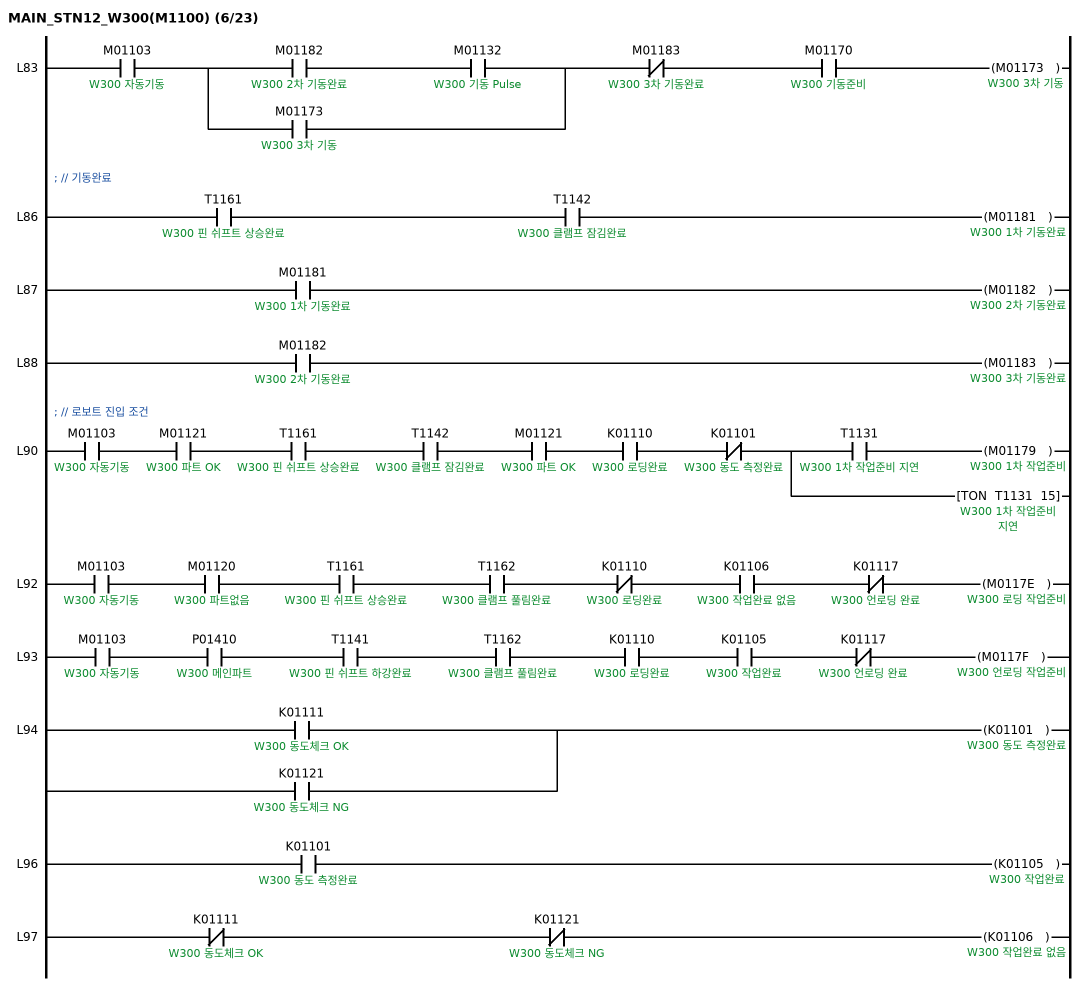
[picture p192: MAIN_STN12_W300(M1100) rungs L83-L97]
; L83
LOAD      M01103	// W300 자동기동
LOAD      M01182	// W300 2차 기동완료
AND       M01132	// W300 기동 Pulse
OR        M01173	// W300 3차 기동
AND LOAD
AND NOT   M01183	// W300 3차 기동완료
AND       M01170	// W300 기동준비
OUT       M01173	// W300 3차 기동
//   // 기동완료
; L86
LOAD      T1161	// W300 핀 쉬프트 상승완료
AND       T1142	// W300 클램프 잠김완료
OUT       M01181	// W300 1차 기동완료
; L87
LOAD      M01181	// W300 1차 기동완료
OUT       M01182	// W300 2차 기동완료
; L88
LOAD      M01182	// W300 2차 기동완료
OUT       M01183	// W300 3차 기동완료
//   // 로보트 진입 조건
; L90
LOAD      M01103	// W300 자동기동
AND       M01121	// W300 파트 OK
AND       T1161	// W300 핀 쉬프트 상승완료
AND       T1142	// W300 클램프 잠김완료
AND       M01121	// W300 파트 OK
AND       K01110	// W300 로딩완료
AND NOT   K01101	// W300 동도 측정완료
MPUSH
AND       T1131	// W300 1차 작업준비 지연
OUT       M01179	// W300 1차 작업준비
MPOP
TON       T1131 15	// W300 1차 작업준비 지연
; L92
LOAD      M01103	// W300 자동기동
AND       M01120	// W300 파트없음
AND       T1161	// W300 핀 쉬프트 상승완료
AND       T1162	// W300 클램프 풀림완료
AND NOT   K01110	// W300 로딩완료
AND       K01106	// W300 작업완료 없음
AND NOT   K01117	// W300 언로딩 완료
OUT       M0117E	// W300 로딩 작업준비
; L93
LOAD      M01103	// W300 자동기동
AND       P01410	// W300 메인파트
AND       T1141	// W300 핀 쉬프트 하강완료
AND       T1162	// W300 클램프 풀림완료
AND       K01110	// W300 로딩완료
AND       K01105	// W300 작업완료
AND NOT   K01117	// W300 언로딩 완료
OUT       M0117F	// W300 언로딩 작업준비
; L94
LOAD      K01111	// W300 동도체크 OK
OR        K01121	// W300 동도체크 NG
OUT       K01101	// W300 동도 측정완료
; L96
LOAD      K01101	// W300 동도 측정완료
OUT       K01105	// W300 작업완료
; L97
LOAD NOT  K01111	// W300 동도체크 OK
AND NOT   K01121	// W300 동도체크 NG
OUT       K01106	// W300 작업완료 없음

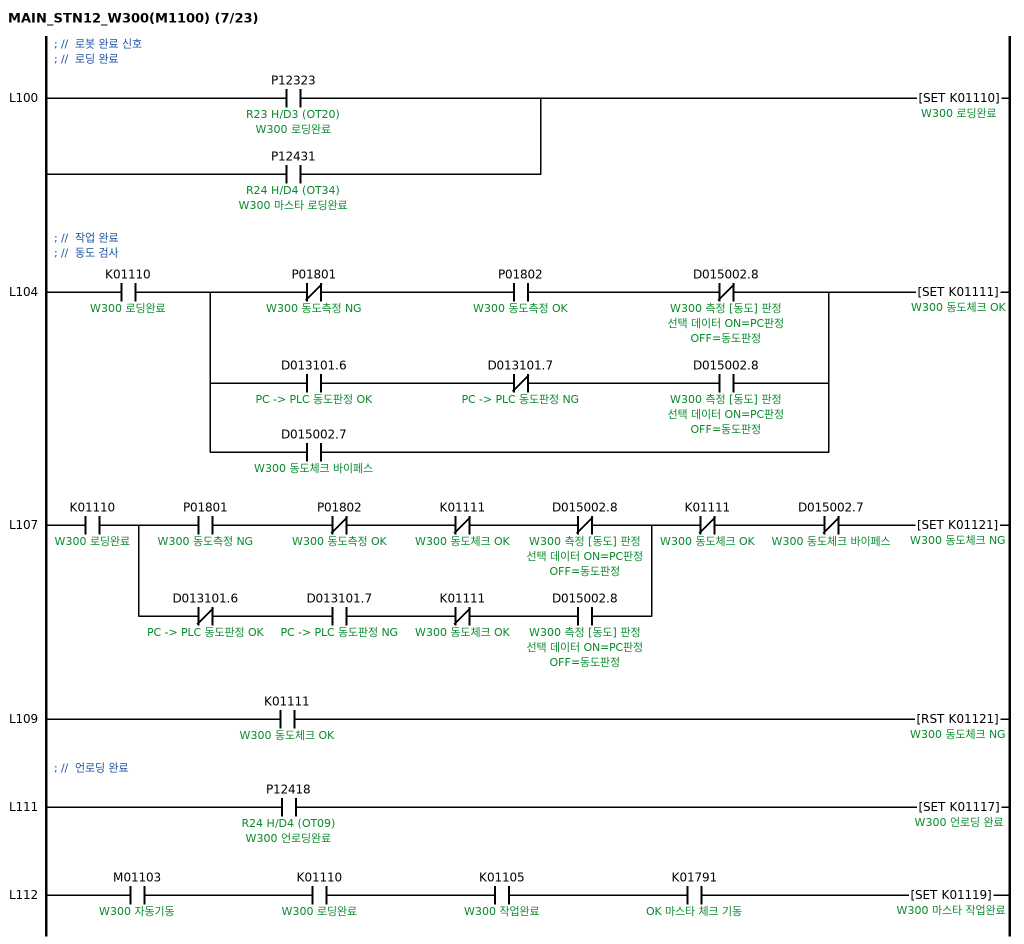
//   //  로봇 완료 신호
//   //  로딩 완료
; L100
LOAD      P12323	// R23 H/D3 (OT20) W300 로딩완료
OR        P12431	// R24 H/D4 (OT34) W300 마스타 로딩완료
SET       K01110	// W300 로딩완료
//   //  작업 완료
//   //  동도 검사
; L104
LOAD      K01110	// W300 로딩완료
LOAD NOT  P01801	// W300 동도측정 NG
AND       P01802	// W300 동도측정 OK
AND NOT   D015002.8	// W300 측정 [동도] 판정 선택 데이터 ON=PC판정 OFF=동도판정
LOAD      D013101.6	// PC -> PLC 동도판정 OK
AND NOT   D013101.7	// PC -> PLC 동도판정 NG
AND       D015002.8	// W300 측정 [동도] 판정 선택 데이터 ON=PC판정 OFF=동도판정
OR LOAD
OR        D015002.7	// W300 동도체크 바이페스
AND LOAD
SET       K01111	// W300 동도체크 OK
; L107
LOAD      K01110	// W300 로딩완료
LOAD      P01801	// W300 동도측정 NG
AND NOT   P01802	// W300 동도측정 OK
AND NOT   K01111	// W300 동도체크 OK
AND NOT   D015002.8	// W300 측정 [동도] 판정 선택 데이터 ON=PC판정 OFF=동도판정
LOAD NOT  D013101.6	// PC -> PLC 동도판정 OK
AND       D013101.7	// PC -> PLC 동도판정 NG
AND NOT   K01111	// W300 동도체크 OK
AND       D015002.8	// W300 측정 [동도] 판정 선택 데이터 ON=PC판정 OFF=동도판정
OR LOAD
AND LOAD
AND NOT   K01111	// W300 동도체크 OK
AND NOT   D015002.7	// W300 동도체크 바이페스
SET       K01121	// W300 동도체크 NG
; L109
LOAD      K01111	// W300 동도체크 OK
RST       K01121	// W300 동도체크 NG
//   //  언로딩 완료
; L111
LOAD      P12418	// R24 H/D4 (OT09) W300 언로딩완료
SET       K01117	// W300 언로딩 완료
; L112
LOAD      M01103	// W300 자동기동
AND       K01110	// W300 로딩완료
AND       K01105	// W300 작업완료
AND       K01791	// OK 마스타 체크 기동
SET       K01119	// W300 마스타 작업완료

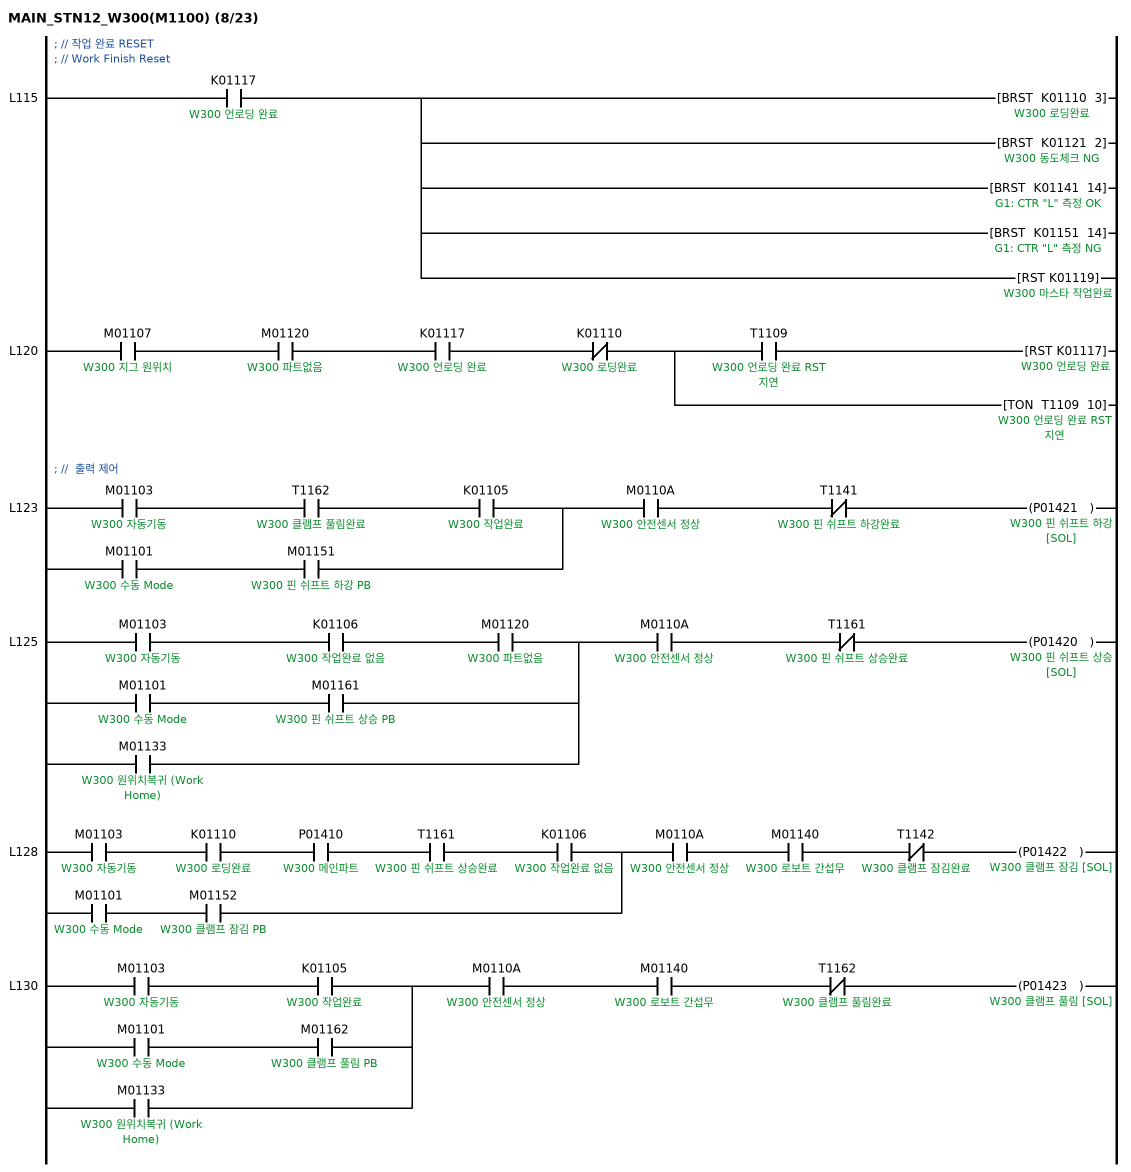
//     // 작업 완료 RESET
//   // Work Finish Reset
; L115
LOAD      K01117	// W300 언로딩 완료
BRST      K01110 3	// W300 로딩완료
BRST      K01121 2	// W300 동도체크 NG
BRST      K01141 14	// G1: CTR "L" 측정 OK
BRST      K01151 14	// G1: CTR "L" 측정 NG
RST       K01119	// W300 마스타 작업완료
; L120
LOAD      M01107	// W300 지그 원위치
AND       M01120	// W300 파트없음
AND       K01117	// W300 언로딩 완료
AND NOT   K01110	// W300 로딩완료
MPUSH
AND       T1109	// W300 언로딩 완료 RST 지연
RST       K01117	// W300 언로딩 완료
MPOP
TON       T1109 10	// W300 언로딩 완료 RST 지연
//     //  출력 제어
; L123
LOAD      M01103	// W300 자동기동
AND       T1162	// W300 클램프 풀림완료
AND       K01105	// W300 작업완료
LOAD      M01101	// W300 수동 Mode
AND       M01151	// W300 핀 쉬프트 하강 PB
OR LOAD
AND       M0110A	// W300 안전센서 정상
AND NOT   T1141	// W300 핀 쉬프트 하강완료
OUT       P01421	// W300 핀 쉬프트 하강 [SOL]
; L125
LOAD      M01103	// W300 자동기동
AND       K01106	// W300 작업완료 없음
AND       M01120	// W300 파트없음
LOAD      M01101	// W300 수동 Mode
AND       M01161	// W300 핀 쉬프트 상승 PB
OR LOAD
OR        M01133	// W300 원위치복귀 (Work Home)
AND       M0110A	// W300 안전센서 정상
AND NOT   T1161	// W300 핀 쉬프트 상승완료
OUT       P01420	// W300 핀 쉬프트 상승 [SOL]
; L128
LOAD      M01103	// W300 자동기동
AND       K01110	// W300 로딩완료
AND       P01410	// W300 메인파트
AND       T1161	// W300 핀 쉬프트 상승완료
AND       K01106	// W300 작업완료 없음
LOAD      M01101	// W300 수동 Mode
AND       M01152	// W300 클램프 잠김 PB
OR LOAD
AND       M0110A	// W300 안전센서 정상
AND       M01140	// W300 로보트 간섭무
AND NOT   T1142	// W300 클램프 잠김완료
OUT       P01422	// W300 클램프 잠김 [SOL]
; L130
LOAD      M01103	// W300 자동기동
AND       K01105	// W300 작업완료
LOAD      M01101	// W300 수동 Mode
AND       M01162	// W300 클램프 풀림 PB
OR LOAD
OR        M01133	// W300 원위치복귀 (Work Home)
AND       M0110A	// W300 안전센서 정상
AND       M01140	// W300 로보트 간섭무
AND NOT   T1162	// W300 클램프 풀림완료
OUT       P01423	// W300 클램프 풀림 [SOL]

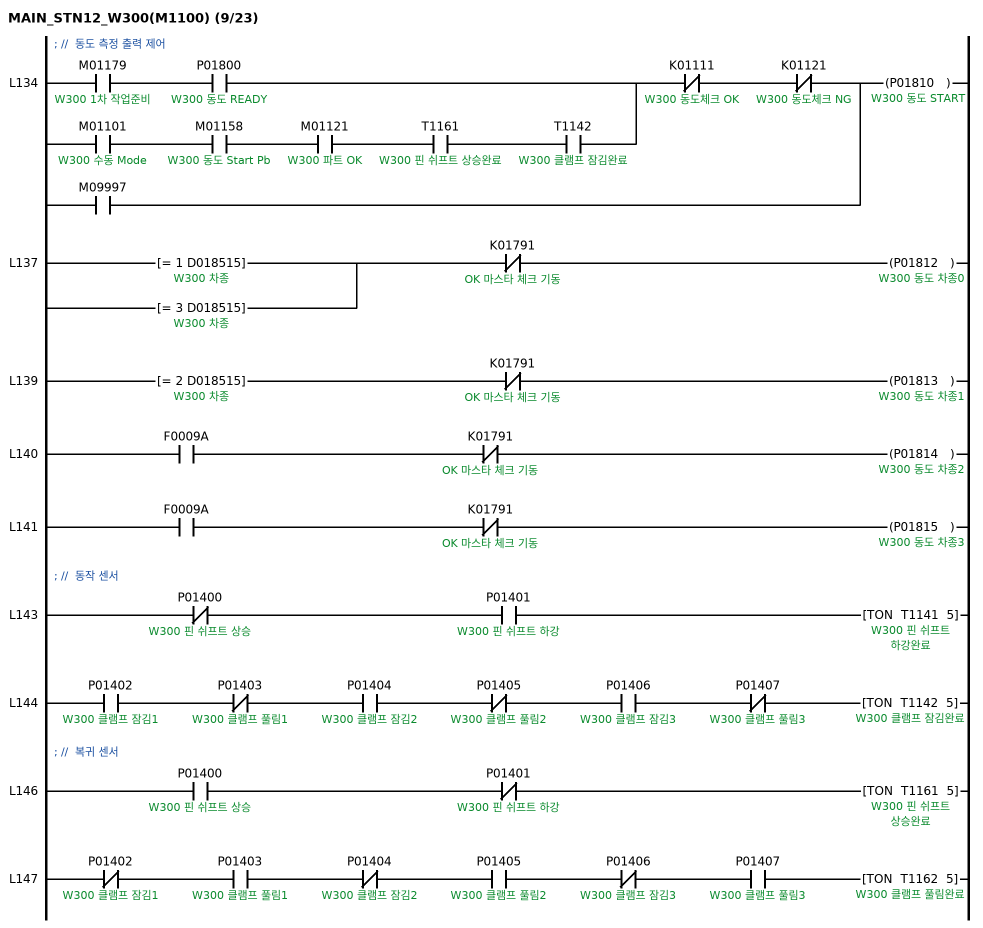
//   //  동도 측정 출력 제어
; L134
LOAD      M01179	// W300 1차 작업준비
AND       P01800	// W300 동도 READY
LOAD      M01101	// W300 수동 Mode
AND       M01158	// W300 동도 Start Pb
AND       M01121	// W300 파트 OK
AND       T1161	// W300 핀 쉬프트 상승완료
AND       T1142	// W300 클램프 잠김완료
OR LOAD
AND NOT   K01111	// W300 동도체크 OK
AND NOT   K01121	// W300 동도체크 NG
OR        M09997
OUT       P01810	// W300 동도 START
; L137
LOAD=     1 D018515	// W300 차종
OR=       3 D018515	// W300 차종
AND NOT   K01791	// OK 마스타 체크 기동
OUT       P01812	// W300 동도 차종0
; L139
LOAD=     2 D018515	// W300 차종
AND NOT   K01791	// OK 마스타 체크 기동
OUT       P01813	// W300 동도 차종1
; L140
LOAD      F0009A
AND NOT   K01791	// OK 마스타 체크 기동
OUT       P01814	// W300 동도 차종2
; L141
LOAD      F0009A
AND NOT   K01791	// OK 마스타 체크 기동
OUT       P01815	// W300 동도 차종3
//   //  동작 센서
; L143
LOAD NOT  P01400	// W300 핀 쉬프트 상승
AND       P01401	// W300 핀 쉬프트 하강
TON       T1141 5	// W300 핀 쉬프트 하강완료
; L144
LOAD      P01402	// W300 클램프 잠김1
AND NOT   P01403	// W300 클램프 풀림1
AND       P01404	// W300 클램프 잠김2
AND NOT   P01405	// W300 클램프 풀림2
AND       P01406	// W300 클램프 잠김3
AND NOT   P01407	// W300 클램프 풀림3
TON       T1142 5	// W300 클램프 잠김완료
//   //  복귀 센서
; L146
LOAD      P01400	// W300 핀 쉬프트 상승
AND NOT   P01401	// W300 핀 쉬프트 하강
TON       T1161 5	// W300 핀 쉬프트 상승완료
; L147
LOAD NOT  P01402	// W300 클램프 잠김1
AND       P01403	// W300 클램프 풀림1
AND NOT   P01404	// W300 클램프 잠김2
AND       P01405	// W300 클램프 풀림2
AND NOT   P01406	// W300 클램프 잠김3
AND       P01407	// W300 클램프 풀림3
TON       T1162 5	// W300 클램프 풀림완료

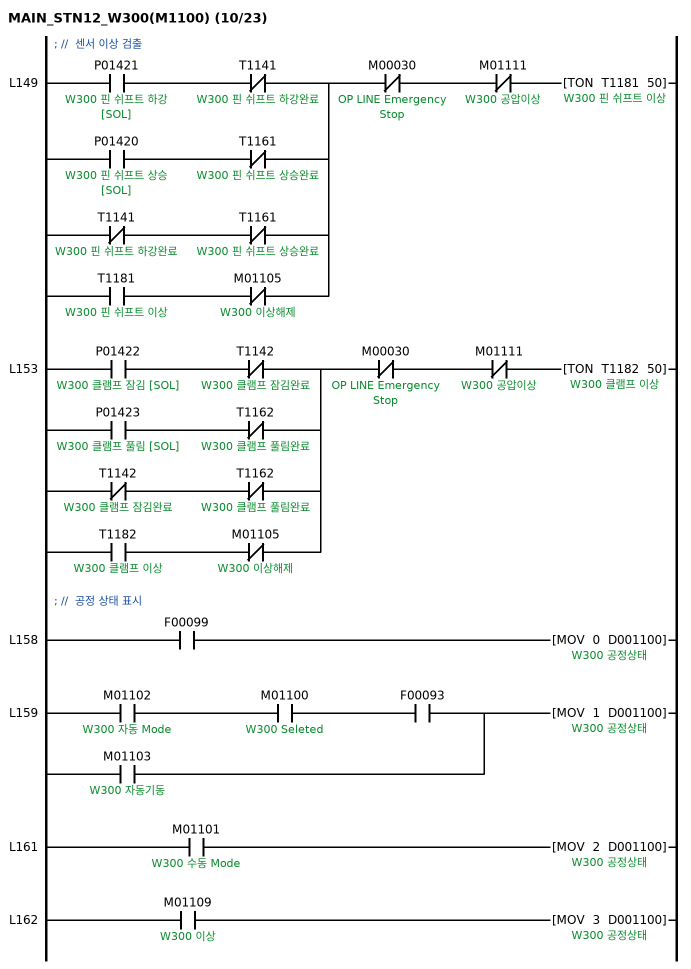
//     //  센서 이상 검출
; L149
LOAD      P01421	// W300 핀 쉬프트 하강 [SOL]
AND NOT   T1141	// W300 핀 쉬프트 하강완료
LOAD      P01420	// W300 핀 쉬프트 상승 [SOL]
AND NOT   T1161	// W300 핀 쉬프트 상승완료
OR LOAD
LOAD NOT  T1141	// W300 핀 쉬프트 하강완료
AND NOT   T1161	// W300 핀 쉬프트 상승완료
OR LOAD
LOAD      T1181	// W300 핀 쉬프트 이상
AND NOT   M01105	// W300 이상해제
OR LOAD
AND NOT   M00030	// OP LINE Emergency Stop
AND NOT   M01111	// W300 공압이상
TON       T1181 50	// W300 핀 쉬프트 이상
; L153
LOAD      P01422	// W300 클램프 잠김 [SOL]
AND NOT   T1142	// W300 클램프 잠김완료
LOAD      P01423	// W300 클램프 풀림 [SOL]
AND NOT   T1162	// W300 클램프 풀림완료
OR LOAD
LOAD NOT  T1142	// W300 클램프 잠김완료
AND NOT   T1162	// W300 클램프 풀림완료
OR LOAD
LOAD      T1182	// W300 클램프 이상
AND NOT   M01105	// W300 이상해제
OR LOAD
AND NOT   M00030	// OP LINE Emergency Stop
AND NOT   M01111	// W300 공압이상
TON       T1182 50	// W300 클램프 이상
//   //  공정 상태 표시
; L158
LOAD      F00099
MOV       0 D001100	// W300 공정상태
; L159
LOAD      M01102	// W300 자동 Mode
AND       M01100	// W300 Seleted
AND       F00093
OR        M01103	// W300 자동기동
MOV       1 D001100	// W300 공정상태
; L161
LOAD      M01101	// W300 수동 Mode
MOV       2 D001100	// W300 공정상태
; L162
LOAD      M01109	// W300 이상
MOV       3 D001100	// W300 공정상태

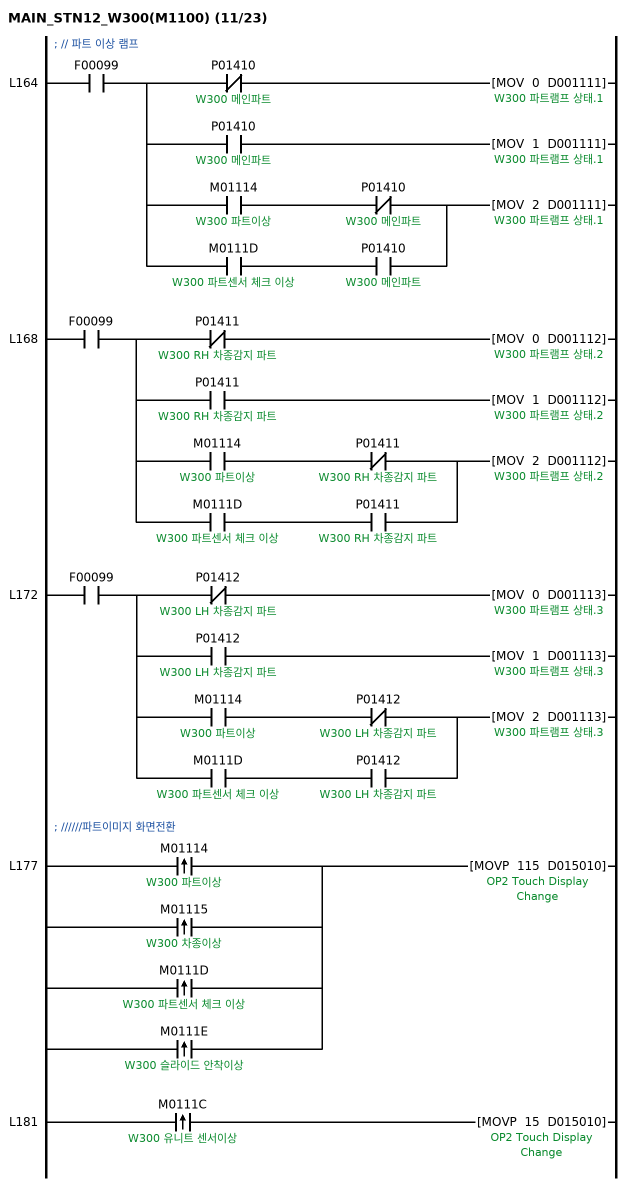
//   // 파트 이상 램프
; L164
LOAD      F00099
MPUSH
AND NOT   P01410	// W300 메인파트
MOV       0 D001111	// W300 파트램프 상태.1
MLOAD
AND       P01410	// W300 메인파트
MOV       1 D001111	// W300 파트램프 상태.1
MPOP
LOAD      M01114	// W300 파트이상
AND NOT   P01410	// W300 메인파트
LOAD      M0111D	// W300 파트센서 체크 이상
AND       P01410	// W300 메인파트
OR LOAD
AND LOAD
MOV       2 D001111	// W300 파트램프 상태.1
; L168
LOAD      F00099
MPUSH
AND NOT   P01411	// W300 RH 차종감지 파트
MOV       0 D001112	// W300 파트램프 상태.2
MLOAD
AND       P01411	// W300 RH 차종감지 파트
MOV       1 D001112	// W300 파트램프 상태.2
MPOP
LOAD      M01114	// W300 파트이상
AND NOT   P01411	// W300 RH 차종감지 파트
LOAD      M0111D	// W300 파트센서 체크 이상
AND       P01411	// W300 RH 차종감지 파트
OR LOAD
AND LOAD
MOV       2 D001112	// W300 파트램프 상태.2
; L172
LOAD      F00099
MPUSH
AND NOT   P01412	// W300 LH 차종감지 파트
MOV       0 D001113	// W300 파트램프 상태.3
MLOAD
AND       P01412	// W300 LH 차종감지 파트
MOV       1 D001113	// W300 파트램프 상태.3
MPOP
LOAD      M01114	// W300 파트이상
AND NOT   P01412	// W300 LH 차종감지 파트
LOAD      M0111D	// W300 파트센서 체크 이상
AND       P01412	// W300 LH 차종감지 파트
OR LOAD
AND LOAD
MOV       2 D001113	// W300 파트램프 상태.3
// //////파트이미지 화면전환
; L177
LOADP     M01114	// W300 파트이상
ORP       M01115	// W300 차종이상
ORP       M0111D	// W300 파트센서 체크 이상
ORP       M0111E	// W300 슬라이드 안착이상
MOVP      115 D015010	// OP2 Touch Display Change
; L181
LOADP     M0111C	// W300 유니트 센서이상
MOVP      15 D015010	// OP2 Touch Display Change

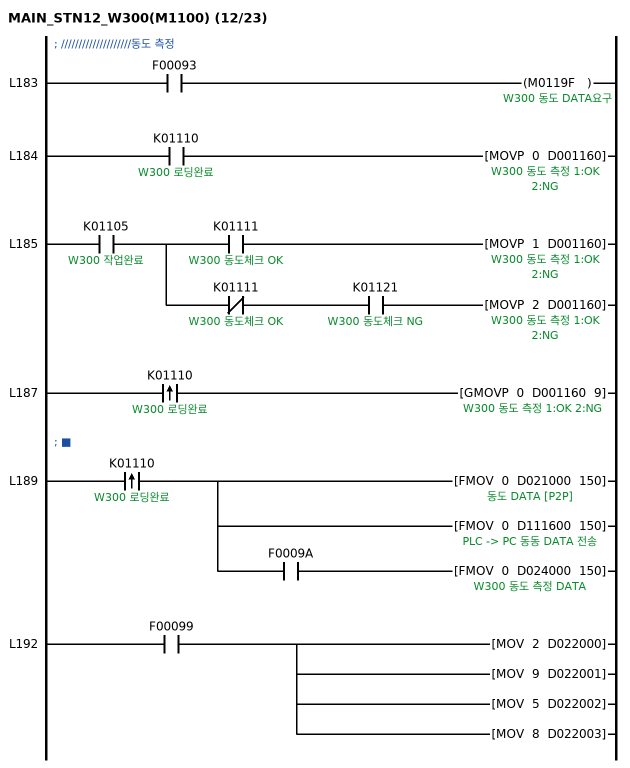
// ////////////////////동도 측정
; L183
LOAD      F00093
OUT       M0119F	// W300 동도 DATA요구
; L184
LOAD      K01110	// W300 로딩완료
MOVP      0 D001160	// W300 동도 측정 1:OK 2:NG
; L185
LOAD      K01105	// W300 작업완료
MPUSH
AND       K01111	// W300 동도체크 OK
MOVP      1 D001160	// W300 동도 측정 1:OK 2:NG
MPOP
AND NOT   K01111	// W300 동도체크 OK
AND       K01121	// W300 동도체크 NG
MOVP      2 D001160	// W300 동도 측정 1:OK 2:NG
; L187
LOADP     K01110	// W300 로딩완료
GMOVP     0 D001160 9	// W300 동도 측정 1:OK 2:NG
//  ■
; L189
LOADP     K01110	// W300 로딩완료
FMOV      0 D021000 150	// 동도 DATA [P2P]
FMOV      0 D111600 150	// PLC -> PC 동동 DATA 전송
AND       F0009A
FMOV      0 D024000 150	// W300 동도 측정 DATA
; L192
LOAD      F00099
MOV       2 D022000
MOV       9 D022001
MOV       5 D022002
MOV       8 D022003

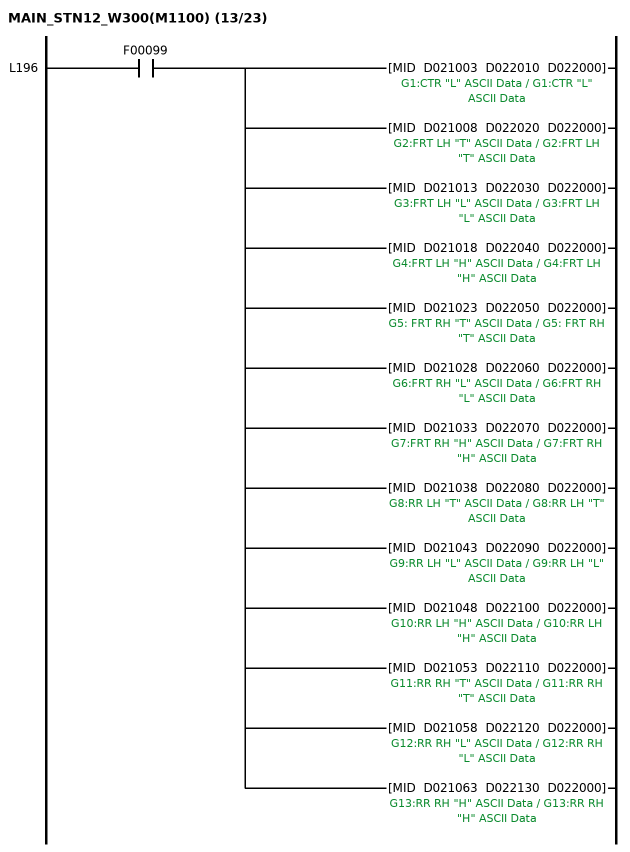
; L196
LOAD      F00099
MID       D021003 D022010 D022000	// G1:CTR "L" ASCII Data / G1:CTR "L" ASCII Data
MID       D021008 D022020 D022000	// G2:FRT LH "T" ASCII Data / G2:FRT LH "T" ASCII Data
MID       D021013 D022030 D022000	// G3:FRT LH "L" ASCII Data / G3:FRT LH "L" ASCII Data
MID       D021018 D022040 D022000	// G4:FRT LH "H" ASCII Data / G4:FRT LH "H" ASCII Data
MID       D021023 D022050 D022000	// G5: FRT RH "T" ASCII Data / G5: FRT RH "T" ASCII Data
MID       D021028 D022060 D022000	// G6:FRT RH "L" ASCII Data / G6:FRT RH "L" ASCII Data
MID       D021033 D022070 D022000	// G7:FRT RH "H" ASCII Data / G7:FRT RH "H" ASCII Data
MID       D021038 D022080 D022000	// G8:RR LH "T" ASCII Data / G8:RR LH "T" ASCII Data
MID       D021043 D022090 D022000	// G9:RR LH "L" ASCII Data / G9:RR LH "L" ASCII Data
MID       D021048 D022100 D022000	// G10:RR LH "H" ASCII Data / G10:RR LH "H" ASCII Data
MID       D021053 D022110 D022000	// G11:RR RH "T" ASCII Data / G11:RR RH "T" ASCII Data
MID       D021058 D022120 D022000	// G12:RR RH "L" ASCII Data / G12:RR RH "L" ASCII Data
MID       D021063 D022130 D022000	// G13:RR RH "H" ASCII Data / G13:RR RH "H" ASCII Data

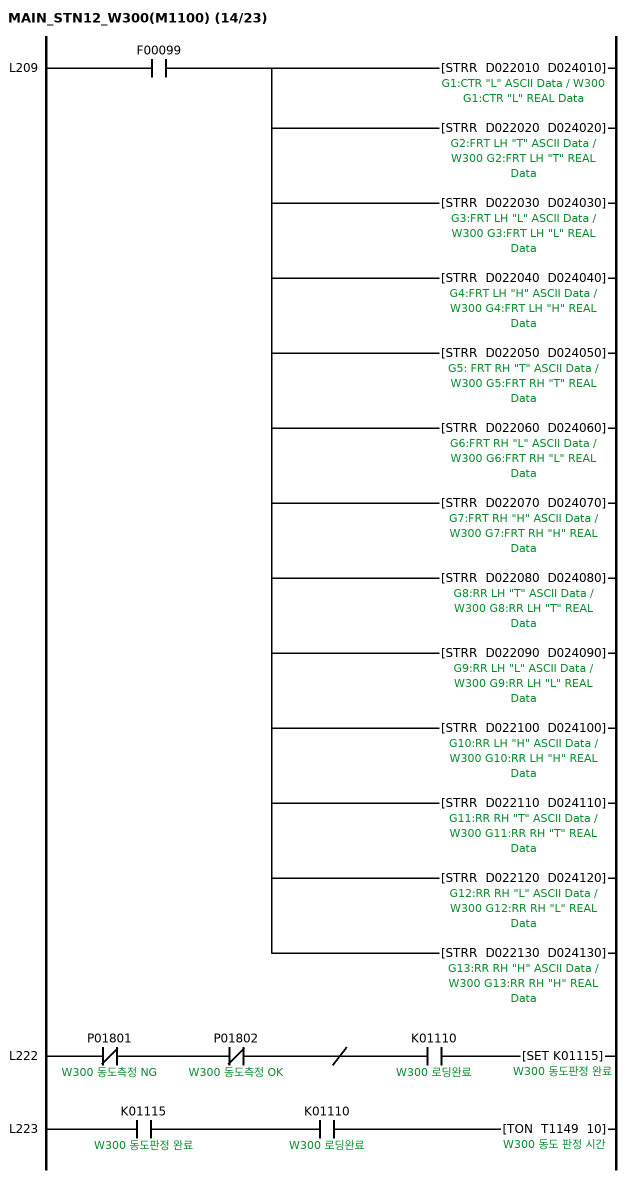
; L209
LOAD      F00099
STRR      D022010 D024010	// G1:CTR "L" ASCII Data / W300 G1:CTR "L" REAL Data
STRR      D022020 D024020	// G2:FRT LH "T" ASCII Data / W300 G2:FRT LH "T" REAL Data
STRR      D022030 D024030	// G3:FRT LH "L" ASCII Data / W300 G3:FRT LH "L" REAL Data
STRR      D022040 D024040	// G4:FRT LH "H" ASCII Data / W300 G4:FRT LH "H" REAL Data
STRR      D022050 D024050	// G5: FRT RH "T" ASCII Data / W300 G5:FRT RH "T" REAL Data
STRR      D022060 D024060	// G6:FRT RH "L" ASCII Data / W300 G6:FRT RH "L" REAL Data
STRR      D022070 D024070	// G7:FRT RH "H" ASCII Data / W300 G7:FRT RH "H" REAL Data
STRR      D022080 D024080	// G8:RR LH "T" ASCII Data / W300 G8:RR LH "T" REAL Data
STRR      D022090 D024090	// G9:RR LH "L" ASCII Data / W300 G9:RR LH "L" REAL Data
STRR      D022100 D024100	// G10:RR LH "H" ASCII Data / W300 G10:RR LH "H" REAL Data
STRR      D022110 D024110	// G11:RR RH "T" ASCII Data / W300 G11:RR RH "T" REAL Data
STRR      D022120 D024120	// G12:RR RH "L" ASCII Data / W300 G12:RR RH "L" REAL Data
STRR      D022130 D024130	// G13:RR RH "H" ASCII Data / W300 G13:RR RH "H" REAL Data
; L222
LOAD NOT  P01801	// W300 동도측정 NG
AND NOT   P01802	// W300 동도측정 OK
NOT
AND       K01110	// W300 로딩완료
SET       K01115	// W300 동도판정 완료
; L223
LOAD      K01115	// W300 동도판정 완료
AND       K01110	// W300 로딩완료
TON       T1149 10	// W300 동도 판정 시간

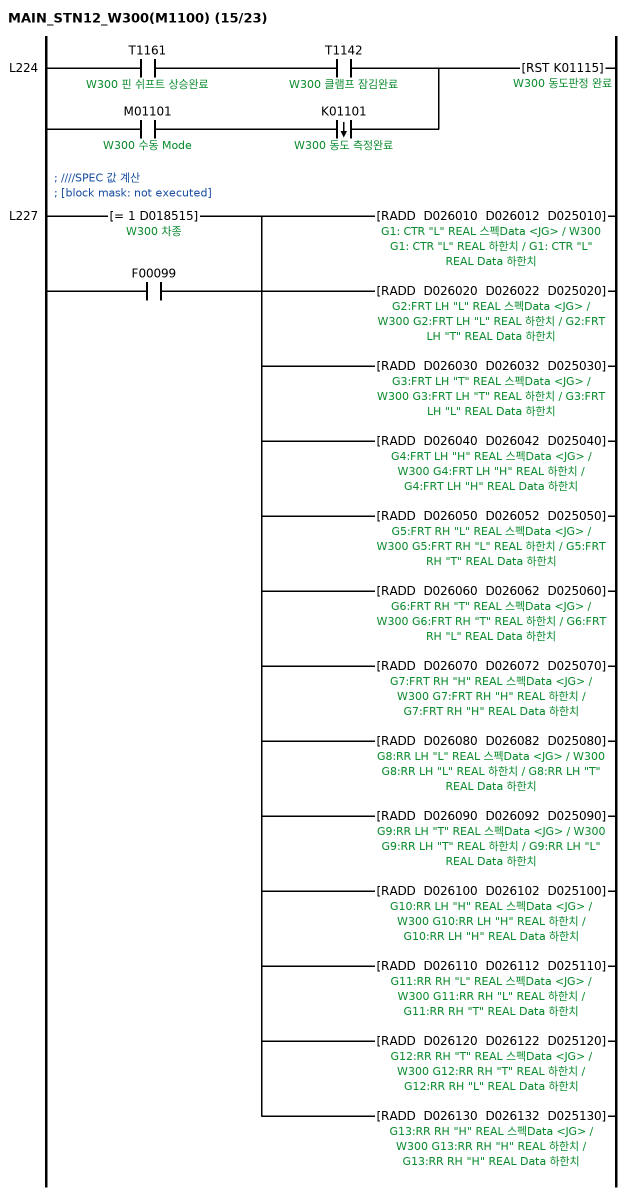
; L224
LOAD      T1161	// W300 핀 쉬프트 상승완료
AND       T1142	// W300 클램프 잠김완료
LOAD      M01101	// W300 수동 Mode
ANDN      K01101	// W300 동도 측정완료
OR LOAD
RST       K01115	// W300 동도판정 완료
// ////SPEC 값 계산
; L227 (block mask: not executed)
LOAD=     1 D018515	// W300 차종
OR        F00099
RADD      D026010 D026012 D025010	// G1: CTR "L" REAL 스펙Data <JG> / W300 G1: CTR "L" REAL 하한치 / G1: CTR "L" REAL Data 하한치
RADD      D026020 D026022 D025020	// G2:FRT LH "L" REAL 스펙Data <JG> / W300 G2:FRT LH "L" REAL 하한치 / G2:FRT LH "T" REAL Data 하한치
RADD      D026030 D026032 D025030	// G3:FRT LH "T" REAL 스펙Data <JG> / W300 G3:FRT LH "T" REAL 하한치 / G3:FRT LH "L" REAL Data 하한치
RADD      D026040 D026042 D025040	// G4:FRT LH "H" REAL 스펙Data <JG> / W300 G4:FRT LH "H" REAL 하한치 / G4:FRT LH "H" REAL Data 하한치
RADD      D026050 D026052 D025050	// G5:FRT RH "L" REAL 스펙Data <JG> / W300 G5:FRT RH "L" REAL 하한치 / G5:FRT RH "T" REAL Data 하한치
RADD      D026060 D026062 D025060	// G6:FRT RH "T" REAL 스펙Data <JG> / W300 G6:FRT RH "T" REAL 하한치 / G6:FRT RH "L" REAL Data 하한치
RADD      D026070 D026072 D025070	// G7:FRT RH "H" REAL 스펙Data <JG> / W300 G7:FRT RH "H" REAL 하한치 / G7:FRT RH "H" REAL Data 하한치
RADD      D026080 D026082 D025080	// G8:RR LH "L" REAL 스펙Data <JG> / W300 G8:RR LH "L" REAL 하한치 / G8:RR LH "T" REAL Data 하한치
RADD      D026090 D026092 D025090	// G9:RR LH "T" REAL 스펙Data <JG> / W300 G9:RR LH "T" REAL 하한치 / G9:RR LH "L" REAL Data 하한치
RADD      D026100 D026102 D025100	// G10:RR LH "H" REAL 스펙Data <JG> / W300 G10:RR LH "H" REAL 하한치 / G10:RR LH "H" REAL Data 하한치
RADD      D026110 D026112 D025110	// G11:RR RH "L" REAL 스펙Data <JG> / W300 G11:RR RH "L" REAL 하한치 / G11:RR RH "T" REAL Data 하한치
RADD      D026120 D026122 D025120	// G12:RR RH "T" REAL 스펙Data <JG> / W300 G12:RR RH "T" REAL 하한치 / G12:RR RH "L" REAL Data 하한치
RADD      D026130 D026132 D025130	// G13:RR RH "H" REAL 스펙Data <JG> / W300 G13:RR RH "H" REAL 하한치 / G13:RR RH "H" REAL Data 하한치

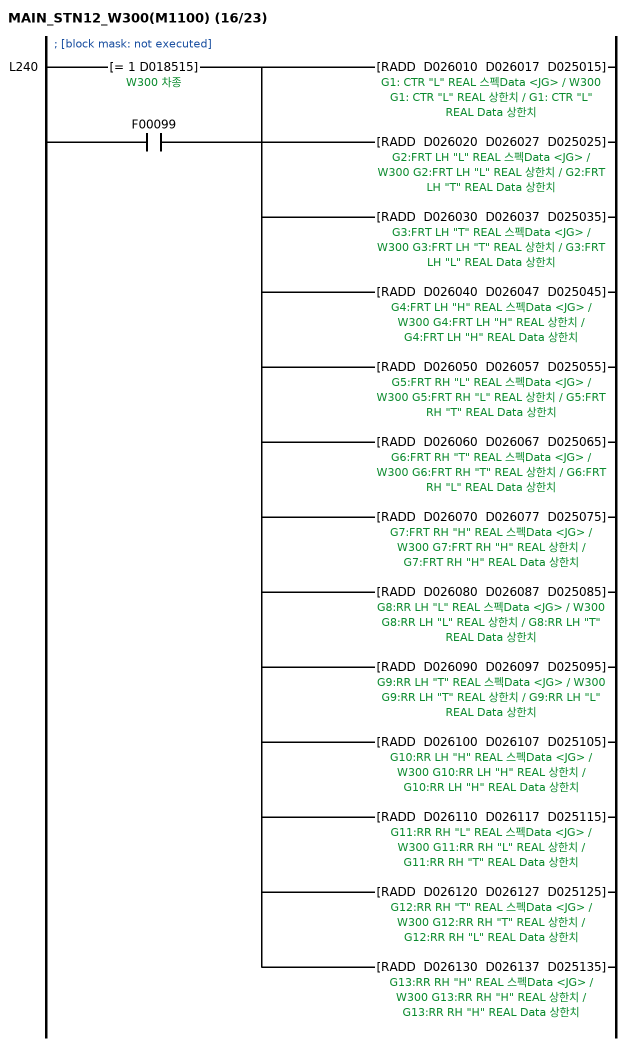
; L240 (block mask: not executed)
LOAD=     1 D018515	// W300 차종
OR        F00099
RADD      D026010 D026017 D025015	// G1: CTR "L" REAL 스펙Data <JG> / W300 G1: CTR "L" REAL 상한치 / G1: CTR "L" REAL Data 상한치
RADD      D026020 D026027 D025025	// G2:FRT LH "L" REAL 스펙Data <JG> / W300 G2:FRT LH "L" REAL 상한치 / G2:FRT LH "T" REAL Data 상한치
RADD      D026030 D026037 D025035	// G3:FRT LH "T" REAL 스펙Data <JG> / W300 G3:FRT LH "T" REAL 상한치 / G3:FRT LH "L" REAL Data 상한치
RADD      D026040 D026047 D025045	// G4:FRT LH "H" REAL 스펙Data <JG> / W300 G4:FRT LH "H" REAL 상한치 / G4:FRT LH "H" REAL Data 상한치
RADD      D026050 D026057 D025055	// G5:FRT RH "L" REAL 스펙Data <JG> / W300 G5:FRT RH "L" REAL 상한치 / G5:FRT RH "T" REAL Data 상한치
RADD      D026060 D026067 D025065	// G6:FRT RH "T" REAL 스펙Data <JG> / W300 G6:FRT RH "T" REAL 상한치 / G6:FRT RH "L" REAL Data 상한치
RADD      D026070 D026077 D025075	// G7:FRT RH "H" REAL 스펙Data <JG> / W300 G7:FRT RH "H" REAL 상한치 / G7:FRT RH "H" REAL Data 상한치
RADD      D026080 D026087 D025085	// G8:RR LH "L" REAL 스펙Data <JG> / W300 G8:RR LH "L" REAL 상한치 / G8:RR LH "T" REAL Data 상한치
RADD      D026090 D026097 D025095	// G9:RR LH "T" REAL 스펙Data <JG> / W300 G9:RR LH "T" REAL 상한치 / G9:RR LH "L" REAL Data 상한치
RADD      D026100 D026107 D025105	// G10:RR LH "H" REAL 스펙Data <JG> / W300 G10:RR LH "H" REAL 상한치 / G10:RR LH "H" REAL Data 상한치
RADD      D026110 D026117 D025115	// G11:RR RH "L" REAL 스펙Data <JG> / W300 G11:RR RH "L" REAL 상한치 / G11:RR RH "T" REAL Data 상한치
RADD      D026120 D026127 D025125	// G12:RR RH "T" REAL 스펙Data <JG> / W300 G12:RR RH "T" REAL 상한치 / G12:RR RH "L" REAL Data 상한치
RADD      D026130 D026137 D025135	// G13:RR RH "H" REAL 스펙Data <JG> / W300 G13:RR RH "H" REAL 상한치 / G13:RR RH "H" REAL Data 상한치

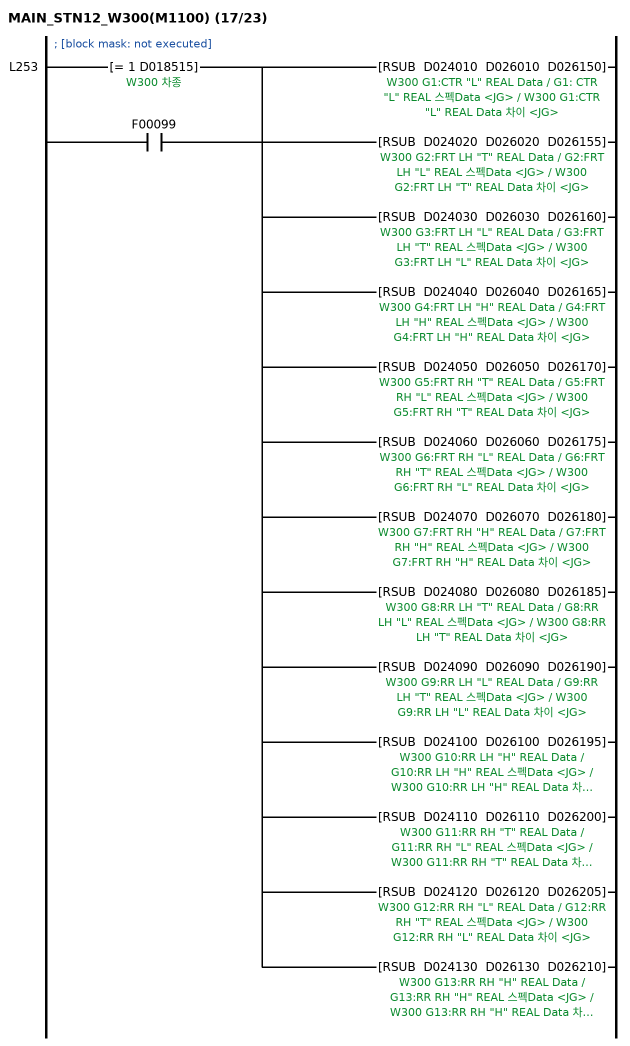
; L253 (block mask: not executed)
LOAD=     1 D018515	// W300 차종
OR        F00099
RSUB      D024010 D026010 D026150	// W300 G1:CTR "L" REAL Data / G1: CTR "L" REAL 스펙Data <JG> / W300 G1:CTR "L" REAL Data 차이 <JG>
RSUB      D024020 D026020 D026155	// W300 G2:FRT LH "T" REAL Data / G2:FRT LH "L" REAL 스펙Data <JG> / W300 G2:FRT LH "T" REAL Data 차이 <JG>
RSUB      D024030 D026030 D026160	// W300 G3:FRT LH "L" REAL Data / G3:FRT LH "T" REAL 스펙Data <JG> / W300 G3:FRT LH "L" REAL Data 차이 <JG>
RSUB      D024040 D026040 D026165	// W300 G4:FRT LH "H" REAL Data / G4:FRT LH "H" REAL 스펙Data <JG> / W300 G4:FRT LH "H" REAL Data 차이 <JG>
RSUB      D024050 D026050 D026170	// W300 G5:FRT RH "T" REAL Data / G5:FRT RH "L" REAL 스펙Data <JG> / W300 G5:FRT RH "T" REAL Data 차이 <JG>
RSUB      D024060 D026060 D026175	// W300 G6:FRT RH "L" REAL Data / G6:FRT RH "T" REAL 스펙Data <JG> / W300 G6:FRT RH "L" REAL Data 차이 <JG>
RSUB      D024070 D026070 D026180	// W300 G7:FRT RH "H" REAL Data / G7:FRT RH "H" REAL 스펙Data <JG> / W300 G7:FRT RH "H" REAL Data 차이 <JG>
RSUB      D024080 D026080 D026185	// W300 G8:RR LH "T" REAL Data / G8:RR LH "L" REAL 스펙Data <JG> / W300 G8:RR LH "T" REAL Data 차이 <JG>
RSUB      D024090 D026090 D026190	// W300 G9:RR LH "L" REAL Data / G9:RR LH "T" REAL 스펙Data <JG> / W300 G9:RR LH "L" REAL Data 차이 <JG>
RSUB      D024100 D026100 D026195	// W300 G10:RR LH "H" REAL Data / G10:RR LH "H" REAL 스펙Data <JG> / W300 G10:RR LH "H" REAL Data 차이 <JG>
RSUB      D024110 D026110 D026200	// W300 G11:RR RH "T" REAL Data / G11:RR RH "L" REAL 스펙Data <JG> / W300 G11:RR RH "T" REAL Data 차이 <JG>
RSUB      D024120 D026120 D026205	// W300 G12:RR RH "L" REAL Data / G12:RR RH "T" REAL 스펙Data <JG> / W300 G12:RR RH "L" REAL Data 차이 <JG>
RSUB      D024130 D026130 D026210	// W300 G13:RR RH "H" REAL Data / G13:RR RH "H" REAL 스펙Data <JG> / W300 G13:RR RH "H" REAL Data 차이 <JG>

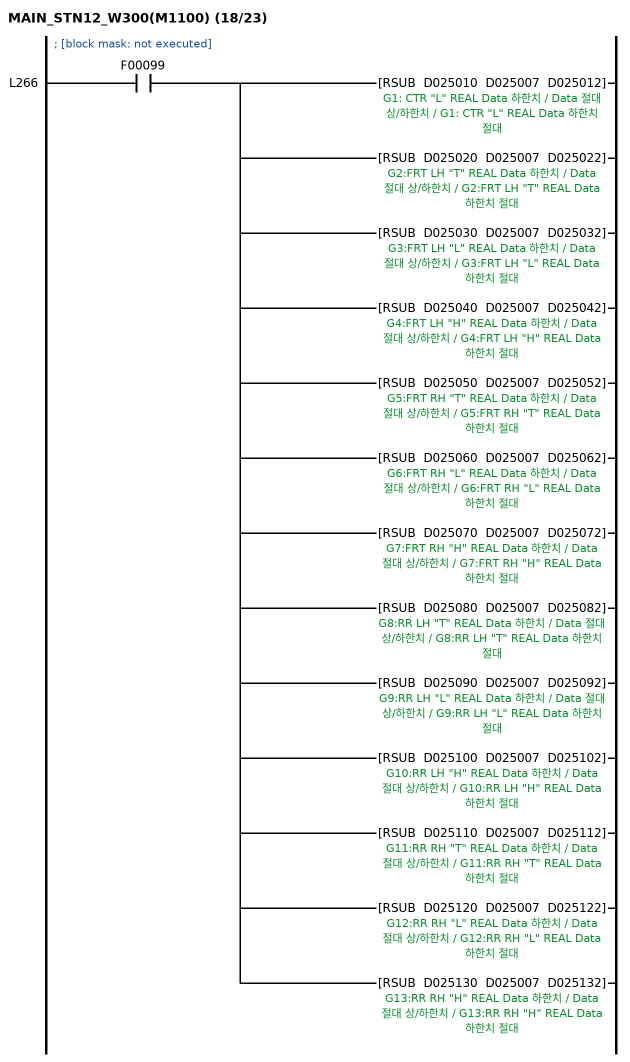
; L266 (block mask: not executed)
LOAD      F00099
RSUB      D025010 D025007 D025012	// G1: CTR "L" REAL Data 하한치 / Data 절대 상/하한치 / G1: CTR "L" REAL Data 하한치 절대
RSUB      D025020 D025007 D025022	// G2:FRT LH "T" REAL Data 하한치 / Data 절대 상/하한치 / G2:FRT LH "T" REAL Data 하한치 절대
RSUB      D025030 D025007 D025032	// G3:FRT LH "L" REAL Data 하한치 / Data 절대 상/하한치 / G3:FRT LH "L" REAL Data 하한치 절대
RSUB      D025040 D025007 D025042	// G4:FRT LH "H" REAL Data 하한치 / Data 절대 상/하한치 / G4:FRT LH "H" REAL Data 하한치 절대
RSUB      D025050 D025007 D025052	// G5:FRT RH "T" REAL Data 하한치 / Data 절대 상/하한치 / G5:FRT RH "T" REAL Data 하한치 절대
RSUB      D025060 D025007 D025062	// G6:FRT RH "L" REAL Data 하한치 / Data 절대 상/하한치 / G6:FRT RH "L" REAL Data 하한치 절대
RSUB      D025070 D025007 D025072	// G7:FRT RH "H" REAL Data 하한치 / Data 절대 상/하한치 / G7:FRT RH "H" REAL Data 하한치 절대
RSUB      D025080 D025007 D025082	// G8:RR LH "T" REAL Data 하한치 / Data 절대 상/하한치 / G8:RR LH "T" REAL Data 하한치 절대
RSUB      D025090 D025007 D025092	// G9:RR LH "L" REAL Data 하한치 / Data 절대 상/하한치 / G9:RR LH "L" REAL Data 하한치 절대
RSUB      D025100 D025007 D025102	// G10:RR LH "H" REAL Data 하한치 / Data 절대 상/하한치 / G10:RR LH "H" REAL Data 하한치 절대
RSUB      D025110 D025007 D025112	// G11:RR RH "T" REAL Data 하한치 / Data 절대 상/하한치 / G11:RR RH "T" REAL Data 하한치 절대
RSUB      D025120 D025007 D025122	// G12:RR RH "L" REAL Data 하한치 / Data 절대 상/하한치 / G12:RR RH "L" REAL Data 하한치 절대
RSUB      D025130 D025007 D025132	// G13:RR RH "H" REAL Data 하한치 / Data 절대 상/하한치 / G13:RR RH "H" REAL Data 하한치 절대

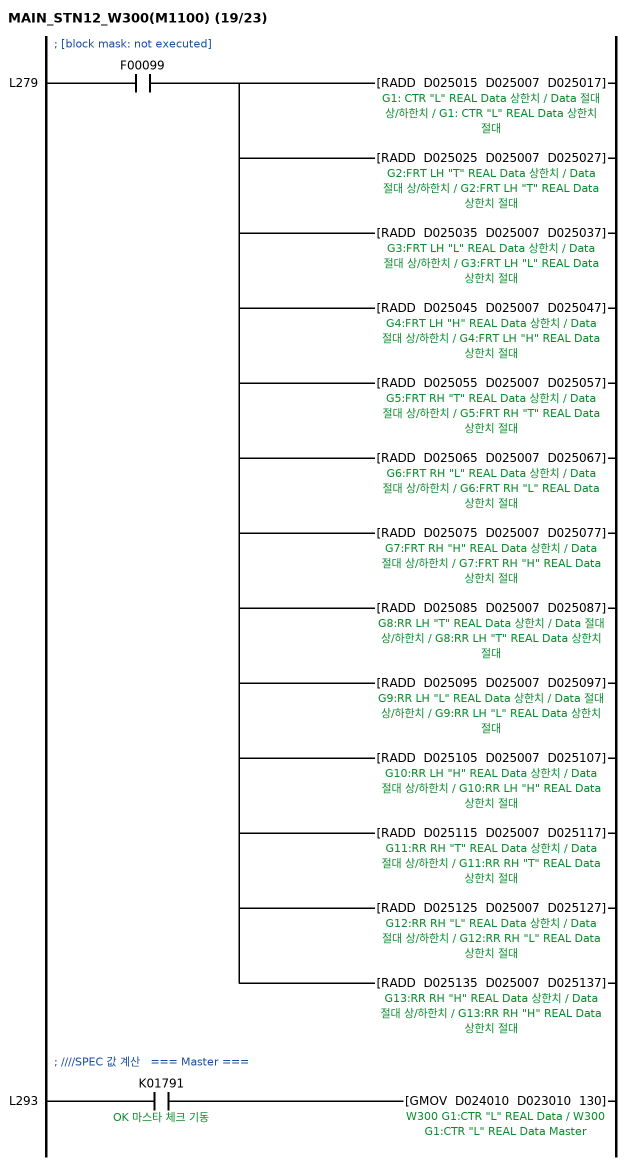
; L279 (block mask: not executed)
LOAD      F00099
RADD      D025015 D025007 D025017	// G1: CTR "L" REAL Data 상한치 / Data 절대 상/하한치 / G1: CTR "L" REAL Data 상한치 절대
RADD      D025025 D025007 D025027	// G2:FRT LH "T" REAL Data 상한치 / Data 절대 상/하한치 / G2:FRT LH "T" REAL Data 상한치 절대
RADD      D025035 D025007 D025037	// G3:FRT LH "L" REAL Data 상한치 / Data 절대 상/하한치 / G3:FRT LH "L" REAL Data 상한치 절대
RADD      D025045 D025007 D025047	// G4:FRT LH "H" REAL Data 상한치 / Data 절대 상/하한치 / G4:FRT LH "H" REAL Data 상한치 절대
RADD      D025055 D025007 D025057	// G5:FRT RH "T" REAL Data 상한치 / Data 절대 상/하한치 / G5:FRT RH "T" REAL Data 상한치 절대
RADD      D025065 D025007 D025067	// G6:FRT RH "L" REAL Data 상한치 / Data 절대 상/하한치 / G6:FRT RH "L" REAL Data 상한치 절대
RADD      D025075 D025007 D025077	// G7:FRT RH "H" REAL Data 상한치 / Data 절대 상/하한치 / G7:FRT RH "H" REAL Data 상한치 절대
RADD      D025085 D025007 D025087	// G8:RR LH "T" REAL Data 상한치 / Data 절대 상/하한치 / G8:RR LH "T" REAL Data 상한치 절대
RADD      D025095 D025007 D025097	// G9:RR LH "L" REAL Data 상한치 / Data 절대 상/하한치 / G9:RR LH "L" REAL Data 상한치 절대
RADD      D025105 D025007 D025107	// G10:RR LH "H" REAL Data 상한치 / Data 절대 상/하한치 / G10:RR LH "H" REAL Data 상한치 절대
RADD      D025115 D025007 D025117	// G11:RR RH "T" REAL Data 상한치 / Data 절대 상/하한치 / G11:RR RH "T" REAL Data 상한치 절대
RADD      D025125 D025007 D025127	// G12:RR RH "L" REAL Data 상한치 / Data 절대 상/하한치 / G12:RR RH "L" REAL Data 상한치 절대
RADD      D025135 D025007 D025137	// G13:RR RH "H" REAL Data 상한치 / Data 절대 상/하한치 / G13:RR RH "H" REAL Data 상한치 절대
// ////SPEC 값 계산   === Master ===
; L293
LOAD      K01791	// OK 마스타 체크 기동
GMOV      D024010 D023010 130	// W300 G1:CTR "L" REAL Data / W300 G1:CTR "L" REAL Data Master

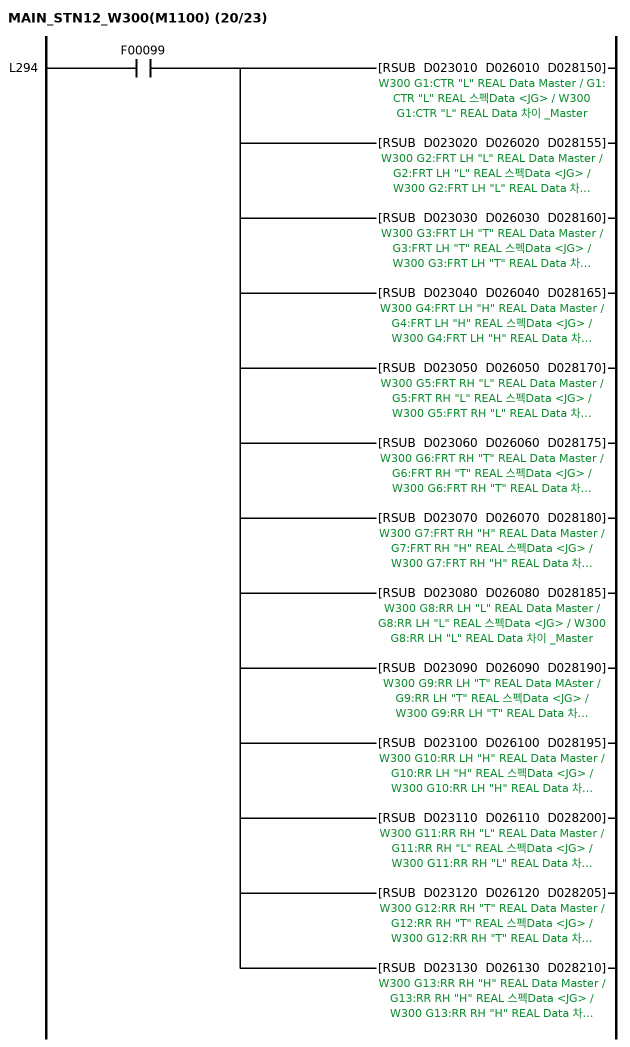
; L294
LOAD      F00099
RSUB      D023010 D026010 D028150	// W300 G1:CTR "L" REAL Data Master / G1: CTR "L" REAL 스펙Data <JG> / W300 G1:CTR "L" REAL Data 차이 _Master
RSUB      D023020 D026020 D028155	// W300 G2:FRT LH "L" REAL Data Master / G2:FRT LH "L" REAL 스펙Data <JG> / W300 G2:FRT LH "L" REAL Data 차이 _Master
RSUB      D023030 D026030 D028160	// W300 G3:FRT LH "T" REAL Data Master / G3:FRT LH "T" REAL 스펙Data <JG> / W300 G3:FRT LH "T" REAL Data 차이 _Master
RSUB      D023040 D026040 D028165	// W300 G4:FRT LH "H" REAL Data Master / G4:FRT LH "H" REAL 스펙Data <JG> / W300 G4:FRT LH "H" REAL Data 차이 _Master
RSUB      D023050 D026050 D028170	// W300 G5:FRT RH "L" REAL Data Master / G5:FRT RH "L" REAL 스펙Data <JG> / W300 G5:FRT RH "L" REAL Data 차이 _Master
RSUB      D023060 D026060 D028175	// W300 G6:FRT RH "T" REAL Data Master / G6:FRT RH "T" REAL 스펙Data <JG> / W300 G6:FRT RH "T" REAL Data 차이 _Master
RSUB      D023070 D026070 D028180	// W300 G7:FRT RH "H" REAL Data Master / G7:FRT RH "H" REAL 스펙Data <JG> / W300 G7:FRT RH "H" REAL Data 차이 _Master
RSUB      D023080 D026080 D028185	// W300 G8:RR LH "L" REAL Data Master / G8:RR LH "L" REAL 스펙Data <JG> / W300 G8:RR LH "L" REAL Data 차이 _Master
RSUB      D023090 D026090 D028190	// W300 G9:RR LH "T" REAL Data MAster / G9:RR LH "T" REAL 스펙Data <JG> / W300 G9:RR LH "T" REAL Data 차이 _Master
RSUB      D023100 D026100 D028195	// W300 G10:RR LH "H" REAL Data Master / G10:RR LH "H" REAL 스펙Data <JG> / W300 G10:RR LH "H" REAL Data 차이 _Master
RSUB      D023110 D026110 D028200	// W300 G11:RR RH "L" REAL Data Master / G11:RR RH "L" REAL 스펙Data <JG> / W300 G11:RR RH "L" REAL Data 차이 _Master
RSUB      D023120 D026120 D028205	// W300 G12:RR RH "T" REAL Data Master / G12:RR RH "T" REAL 스펙Data <JG> / W300 G12:RR RH "T" REAL Data 차이 _Master
RSUB      D023130 D026130 D028210	// W300 G13:RR RH "H" REAL Data Master / G13:RR RH "H" REAL 스펙Data <JG> / W300 G13:RR RH "H" REAL Data 차이 _Master

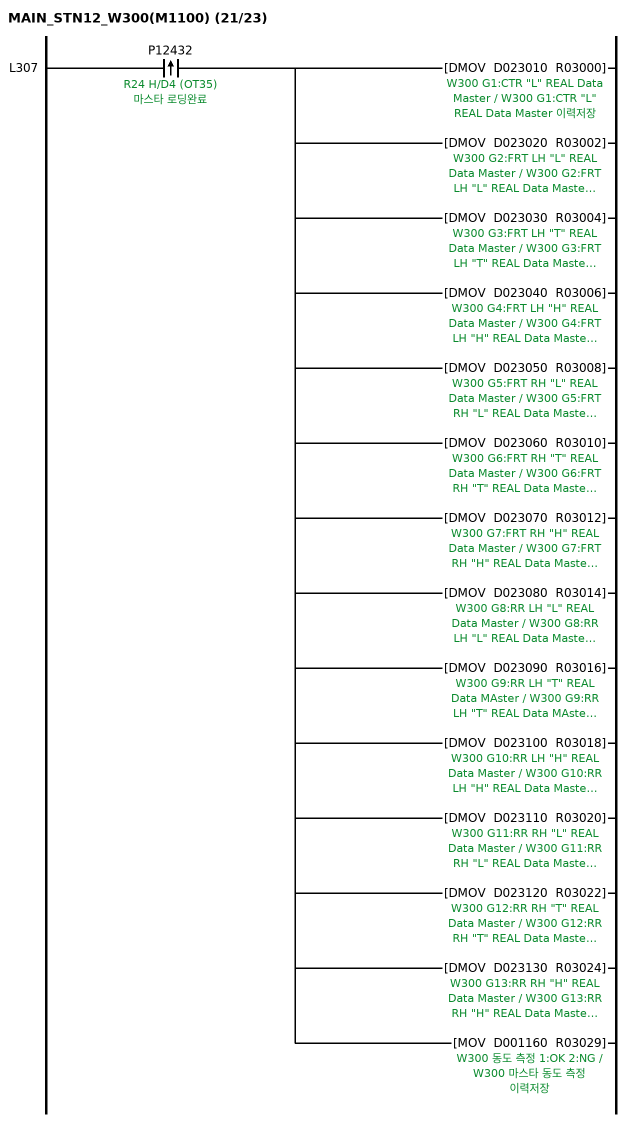
; L307
LOADP     P12432	// R24 H/D4 (OT35) 마스타 로딩완료
DMOV      D023010 R03000	// W300 G1:CTR "L" REAL Data Master / W300 G1:CTR "L" REAL Data Master 이력저장
DMOV      D023020 R03002	// W300 G2:FRT LH "L" REAL Data Master / W300 G2:FRT LH "L" REAL Data Master 이력저장
DMOV      D023030 R03004	// W300 G3:FRT LH "T" REAL Data Master / W300 G3:FRT LH "T" REAL Data Master 이력저장
DMOV      D023040 R03006	// W300 G4:FRT LH "H" REAL Data Master / W300 G4:FRT LH "H" REAL Data Master 이력저장
DMOV      D023050 R03008	// W300 G5:FRT RH "L" REAL Data Master / W300 G5:FRT RH "L" REAL Data Master 이력저장
DMOV      D023060 R03010	// W300 G6:FRT RH "T" REAL Data Master / W300 G6:FRT RH "T" REAL Data Master 이력저장
DMOV      D023070 R03012	// W300 G7:FRT RH "H" REAL Data Master / W300 G7:FRT RH "H" REAL Data Master 이력저장
DMOV      D023080 R03014	// W300 G8:RR LH "L" REAL Data Master / W300 G8:RR LH "L" REAL Data Master 이력저장
DMOV      D023090 R03016	// W300 G9:RR LH "T" REAL Data MAster / W300 G9:RR LH "T" REAL Data MAster 이력저장
DMOV      D023100 R03018	// W300 G10:RR LH "H" REAL Data Master / W300 G10:RR LH "H" REAL Data Master 이력저장
DMOV      D023110 R03020	// W300 G11:RR RH "L" REAL Data Master / W300 G11:RR RH "L" REAL Data Master 이력저장
DMOV      D023120 R03022	// W300 G12:RR RH "T" REAL Data Master / W300 G12:RR RH "T" REAL Data Master 이력저장
DMOV      D023130 R03024	// W300 G13:RR RH "H" REAL Data Master / W300 G13:RR RH "H" REAL Data Master 이력저장
MOV       D001160 R03029	// W300 동도 측정 1:OK 2:NG / W300 마스타 동도 측정 이력저장

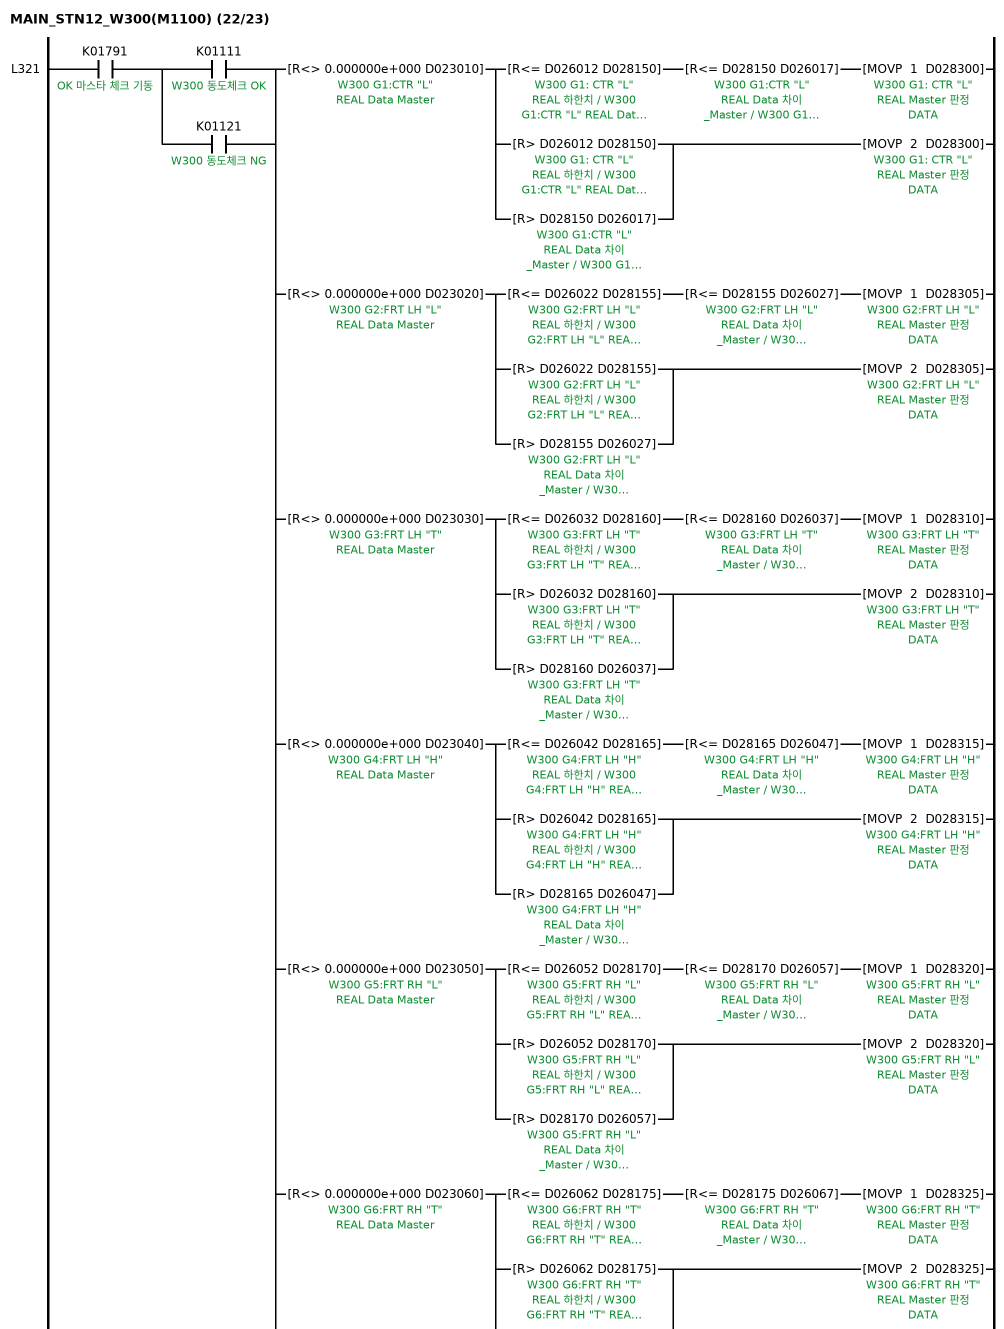

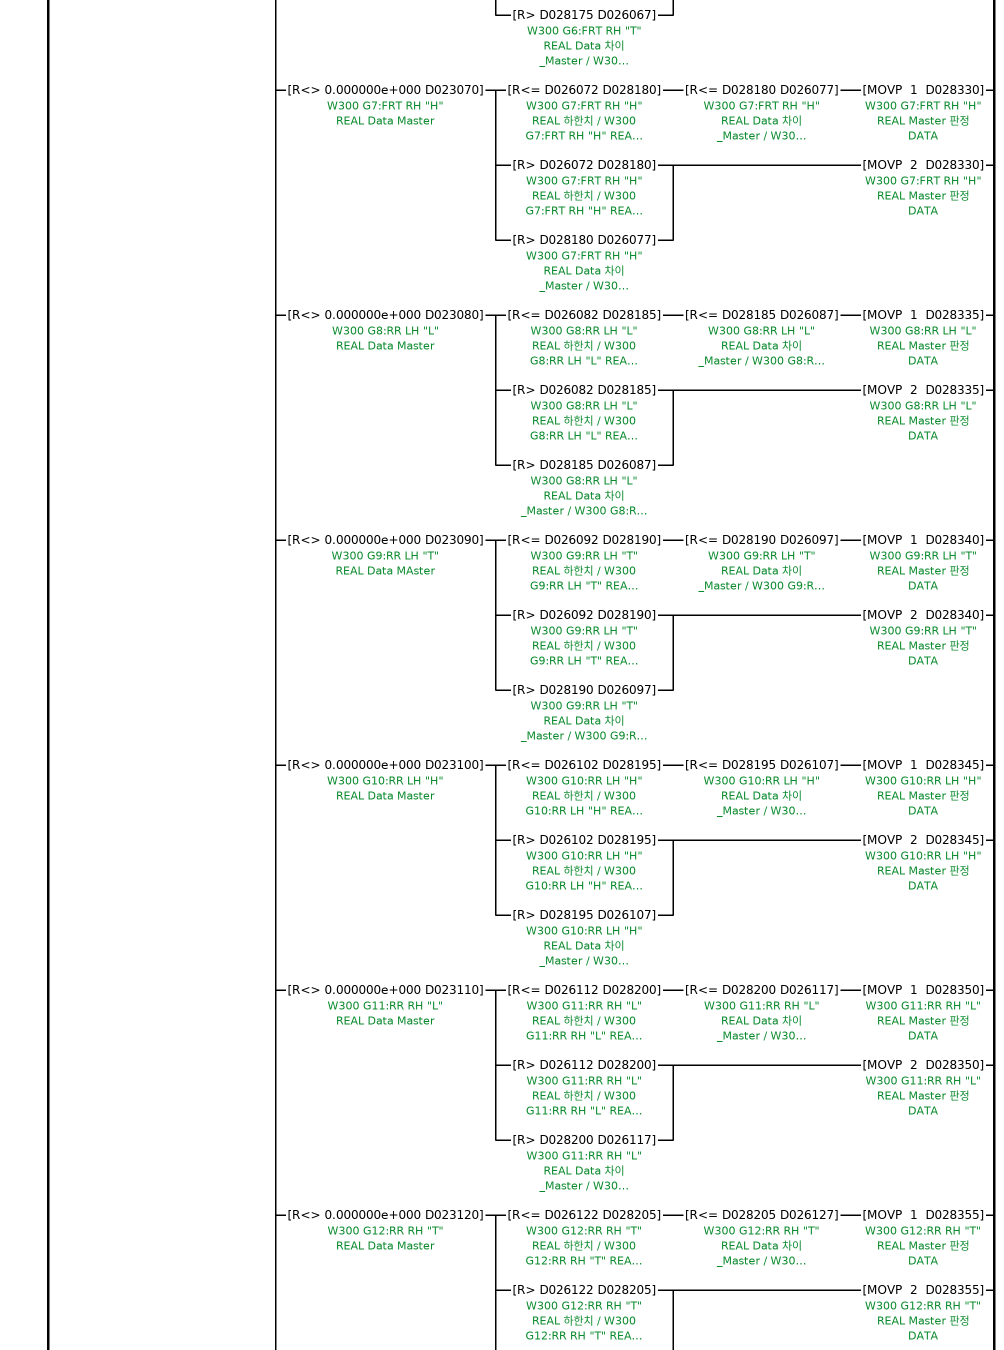

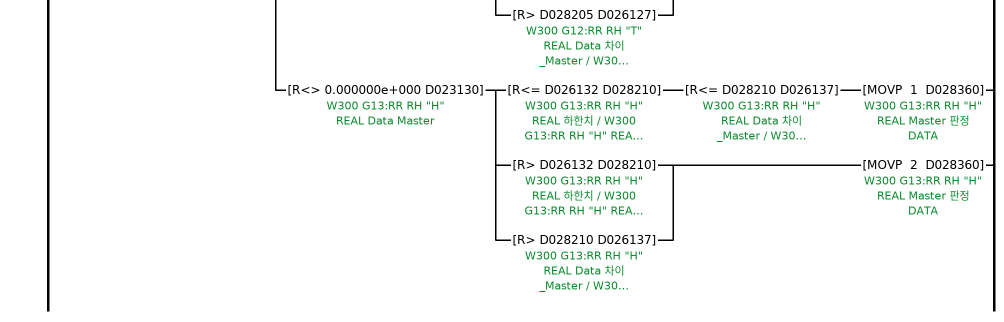
; L321
LOAD      K01791	// OK 마스타 체크 기동
LOAD      K01111	// W300 동도체크 OK
OR        K01121	// W300 동도체크 NG
AND LOAD
MPUSH
ANDR<>    0.000000e+000 D023010	// W300 G1:CTR "L" REAL Data Master
MPUSH
ANDR<=    D026012 D028150	// W300 G1: CTR "L" REAL 하한치 / W300 G1:CTR "L" REAL Data 차이 _Master
ANDR<=    D028150 D026017	// W300 G1:CTR "L" REAL Data 차이 _Master / W300 G1: CTR "L" REAL 상한치
MOVP      1 D028300	// W300 G1: CTR "L" REAL Master 판정 DATA
MPOP
LOADR>    D026012 D028150	// W300 G1: CTR "L" REAL 하한치 / W300 G1:CTR "L" REAL Data 차이 _Master
ORR>      D028150 D026017	// W300 G1:CTR "L" REAL Data 차이 _Master / W300 G1: CTR "L" REAL 상한치
AND LOAD
MOVP      2 D028300	// W300 G1: CTR "L" REAL Master 판정 DATA
MLOAD
ANDR<>    0.000000e+000 D023020	// W300 G2:FRT LH "L" REAL Data Master
MPUSH
ANDR<=    D026022 D028155	// W300 G2:FRT LH "L" REAL 하한치 / W300 G2:FRT LH "L" REAL Data 차이 _Master
ANDR<=    D028155 D026027	// W300 G2:FRT LH "L" REAL Data 차이 _Master / W300 G2:FRT LH "L" REAL 상한치
MOVP      1 D028305	// W300 G2:FRT LH "L" REAL Master 판정 DATA
MPOP
LOADR>    D026022 D028155	// W300 G2:FRT LH "L" REAL 하한치 / W300 G2:FRT LH "L" REAL Data 차이 _Master
ORR>      D028155 D026027	// W300 G2:FRT LH "L" REAL Data 차이 _Master / W300 G2:FRT LH "L" REAL 상한치
AND LOAD
MOVP      2 D028305	// W300 G2:FRT LH "L" REAL Master 판정 DATA
MLOAD
ANDR<>    0.000000e+000 D023030	// W300 G3:FRT LH "T" REAL Data Master
MPUSH
ANDR<=    D026032 D028160	// W300 G3:FRT LH "T" REAL 하한치 / W300 G3:FRT LH "T" REAL Data 차이 _Master
ANDR<=    D028160 D026037	// W300 G3:FRT LH "T" REAL Data 차이 _Master / W300 G3:FRT LH "T" REAL 상한치
MOVP      1 D028310	// W300 G3:FRT LH "T" REAL Master 판정 DATA
MPOP
LOADR>    D026032 D028160	// W300 G3:FRT LH "T" REAL 하한치 / W300 G3:FRT LH "T" REAL Data 차이 _Master
ORR>      D028160 D026037	// W300 G3:FRT LH "T" REAL Data 차이 _Master / W300 G3:FRT LH "T" REAL 상한치
AND LOAD
MOVP      2 D028310	// W300 G3:FRT LH "T" REAL Master 판정 DATA
MLOAD
ANDR<>    0.000000e+000 D023040	// W300 G4:FRT LH "H" REAL Data Master
MPUSH
ANDR<=    D026042 D028165	// W300 G4:FRT LH "H" REAL 하한치 / W300 G4:FRT LH "H" REAL Data 차이 _Master
ANDR<=    D028165 D026047	// W300 G4:FRT LH "H" REAL Data 차이 _Master / W300 G4:FRT LH "H" REAL 상한치
MOVP      1 D028315	// W300 G4:FRT LH "H" REAL Master 판정 DATA
MPOP
LOADR>    D026042 D028165	// W300 G4:FRT LH "H" REAL 하한치 / W300 G4:FRT LH "H" REAL Data 차이 _Master
ORR>      D028165 D026047	// W300 G4:FRT LH "H" REAL Data 차이 _Master / W300 G4:FRT LH "H" REAL 상한치
AND LOAD
MOVP      2 D028315	// W300 G4:FRT LH "H" REAL Master 판정 DATA
MLOAD
ANDR<>    0.000000e+000 D023050	// W300 G5:FRT RH "L" REAL Data Master
MPUSH
ANDR<=    D026052 D028170	// W300 G5:FRT RH "L" REAL 하한치 / W300 G5:FRT RH "L" REAL Data 차이 _Master
ANDR<=    D028170 D026057	// W300 G5:FRT RH "L" REAL Data 차이 _Master / W300 G5:FRT RH "L" REAL 상한치
MOVP      1 D028320	// W300 G5:FRT RH "L" REAL Master 판정 DATA
MPOP
LOADR>    D026052 D028170	// W300 G5:FRT RH "L" REAL 하한치 / W300 G5:FRT RH "L" REAL Data 차이 _Master
ORR>      D028170 D026057	// W300 G5:FRT RH "L" REAL Data 차이 _Master / W300 G5:FRT RH "L" REAL 상한치
AND LOAD
MOVP      2 D028320	// W300 G5:FRT RH "L" REAL Master 판정 DATA
MLOAD
ANDR<>    0.000000e+000 D023060	// W300 G6:FRT RH "T" REAL Data Master
MPUSH
ANDR<=    D026062 D028175	// W300 G6:FRT RH "T" REAL 하한치 / W300 G6:FRT RH "T" REAL Data 차이 _Master
ANDR<=    D028175 D026067	// W300 G6:FRT RH "T" REAL Data 차이 _Master / W300 G6:FRT RH "T" REAL 상한치
MOVP      1 D028325	// W300 G6:FRT RH "T" REAL Master 판정 DATA
MPOP
LOADR>    D026062 D028175	// W300 G6:FRT RH "T" REAL 하한치 / W300 G6:FRT RH "T" REAL Data 차이 _Master
ORR>      D028175 D026067	// W300 G6:FRT RH "T" REAL Data 차이 _Master / W300 G6:FRT RH "T" REAL 상한치
AND LOAD
MOVP      2 D028325	// W300 G6:FRT RH "T" REAL Master 판정 DATA
MLOAD
ANDR<>    0.000000e+000 D023070	// W300 G7:FRT RH "H" REAL Data Master
MPUSH
ANDR<=    D026072 D028180	// W300 G7:FRT RH "H" REAL 하한치 / W300 G7:FRT RH "H" REAL Data 차이 _Master
ANDR<=    D028180 D026077	// W300 G7:FRT RH "H" REAL Data 차이 _Master / W300 G7:FRT RH "H" REAL 상한치
MOVP      1 D028330	// W300 G7:FRT RH "H" REAL Master 판정 DATA
MPOP
LOADR>    D026072 D028180	// W300 G7:FRT RH "H" REAL 하한치 / W300 G7:FRT RH "H" REAL Data 차이 _Master
ORR>      D028180 D026077	// W300 G7:FRT RH "H" REAL Data 차이 _Master / W300 G7:FRT RH "H" REAL 상한치
AND LOAD
MOVP      2 D028330	// W300 G7:FRT RH "H" REAL Master 판정 DATA
MLOAD
ANDR<>    0.000000e+000 D023080	// W300 G8:RR LH "L" REAL Data Master
MPUSH
ANDR<=    D026082 D028185	// W300 G8:RR LH "L" REAL 하한치 / W300 G8:RR LH "L" REAL Data 차이 _Master
ANDR<=    D028185 D026087	// W300 G8:RR LH "L" REAL Data 차이 _Master / W300 G8:RR LH "L" REAL 상한치
MOVP      1 D028335	// W300 G8:RR LH "L" REAL Master 판정 DATA
MPOP
LOADR>    D026082 D028185	// W300 G8:RR LH "L" REAL 하한치 / W300 G8:RR LH "L" REAL Data 차이 _Master
ORR>      D028185 D026087	// W300 G8:RR LH "L" REAL Data 차이 _Master / W300 G8:RR LH "L" REAL 상한치
AND LOAD
MOVP      2 D028335	// W300 G8:RR LH "L" REAL Master 판정 DATA
MLOAD
ANDR<>    0.000000e+000 D023090	// W300 G9:RR LH "T" REAL Data MAster
MPUSH
ANDR<=    D026092 D028190	// W300 G9:RR LH "T" REAL 하한치 / W300 G9:RR LH "T" REAL Data 차이 _Master
ANDR<=    D028190 D026097	// W300 G9:RR LH "T" REAL Data 차이 _Master / W300 G9:RR LH "T" REAL 상한치
MOVP      1 D028340	// W300 G9:RR LH "T" REAL Master 판정 DATA
MPOP
LOADR>    D026092 D028190	// W300 G9:RR LH "T" REAL 하한치 / W300 G9:RR LH "T" REAL Data 차이 _Master
ORR>      D028190 D026097	// W300 G9:RR LH "T" REAL Data 차이 _Master / W300 G9:RR LH "T" REAL 상한치
AND LOAD
MOVP      2 D028340	// W300 G9:RR LH "T" REAL Master 판정 DATA
MLOAD
ANDR<>    0.000000e+000 D023100	// W300 G10:RR LH "H" REAL Data Master
MPUSH
ANDR<=    D026102 D028195	// W300 G10:RR LH "H" REAL 하한치 / W300 G10:RR LH "H" REAL Data 차이 _Master
ANDR<=    D028195 D026107	// W300 G10:RR LH "H" REAL Data 차이 _Master / W300 G10:RR LH "H" REAL 상한치
MOVP      1 D028345	// W300 G10:RR LH "H" REAL Master 판정 DATA
MPOP
LOADR>    D026102 D028195	// W300 G10:RR LH "H" REAL 하한치 / W300 G10:RR LH "H" REAL Data 차이 _Master
ORR>      D028195 D026107	// W300 G10:RR LH "H" REAL Data 차이 _Master / W300 G10:RR LH "H" REAL 상한치
AND LOAD
MOVP      2 D028345	// W300 G10:RR LH "H" REAL Master 판정 DATA
MLOAD
ANDR<>    0.000000e+000 D023110	// W300 G11:RR RH "L" REAL Data Master
MPUSH
ANDR<=    D026112 D028200	// W300 G11:RR RH "L" REAL 하한치 / W300 G11:RR RH "L" REAL Data 차이 _Master
ANDR<=    D028200 D026117	// W300 G11:RR RH "L" REAL Data 차이 _Master / W300 G11:RR RH "L" REAL 상한치
MOVP      1 D028350	// W300 G11:RR RH "L" REAL Master 판정 DATA
MPOP
LOADR>    D026112 D028200	// W300 G11:RR RH "L" REAL 하한치 / W300 G11:RR RH "L" REAL Data 차이 _Master
ORR>      D028200 D026117	// W300 G11:RR RH "L" REAL Data 차이 _Master / W300 G11:RR RH "L" REAL 상한치
AND LOAD
MOVP      2 D028350	// W300 G11:RR RH "L" REAL Master 판정 DATA
MLOAD
ANDR<>    0.000000e+000 D023120	// W300 G12:RR RH "T" REAL Data Master
MPUSH
ANDR<=    D026122 D028205	// W300 G12:RR RH "T" REAL 하한치 / W300 G12:RR RH "T" REAL Data 차이 _Master
ANDR<=    D028205 D026127	// W300 G12:RR RH "T" REAL Data 차이 _Master / W300 G12:RR RH "T" REAL 상한치
MOVP      1 D028355	// W300 G12:RR RH "T" REAL Master 판정 DATA
MPOP
LOADR>    D026122 D028205	// W300 G12:RR RH "T" REAL 하한치 / W300 G12:RR RH "T" REAL Data 차이 _Master
ORR>      D028205 D026127	// W300 G12:RR RH "T" REAL Data 차이 _Master / W300 G12:RR RH "T" REAL 상한치
AND LOAD
MOVP      2 D028355	// W300 G12:RR RH "T" REAL Master 판정 DATA
MPOP
ANDR<>    0.000000e+000 D023130	// W300 G13:RR RH "H" REAL Data Master
MPUSH
ANDR<=    D026132 D028210	// W300 G13:RR RH "H" REAL 하한치 / W300 G13:RR RH "H" REAL Data 차이 _Master
ANDR<=    D028210 D026137	// W300 G13:RR RH "H" REAL Data 차이 _Master / W300 G13:RR RH "H" REAL 상한치
MOVP      1 D028360	// W300 G13:RR RH "H" REAL Master 판정 DATA
MPOP
LOADR>    D026132 D028210	// W300 G13:RR RH "H" REAL 하한치 / W300 G13:RR RH "H" REAL Data 차이 _Master
ORR>      D028210 D026137	// W300 G13:RR RH "H" REAL Data 차이 _Master / W300 G13:RR RH "H" REAL 상한치
AND LOAD
MOVP      2 D028360	// W300 G13:RR RH "H" REAL Master 판정 DATA

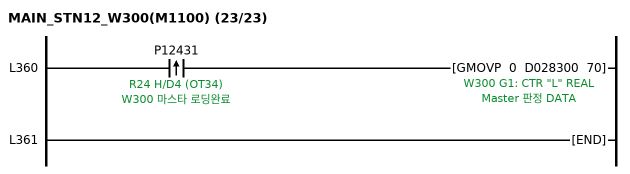
; L360
LOADP     P12431	// R24 H/D4 (OT34) W300 마스타 로딩완료
GMOVP     0 D028300 70	// W300 G1: CTR "L" REAL Master 판정 DATA
; L361
END

PROGRAM MAIN_STN13_W400(M1200) (task: 스캔 프로그램)

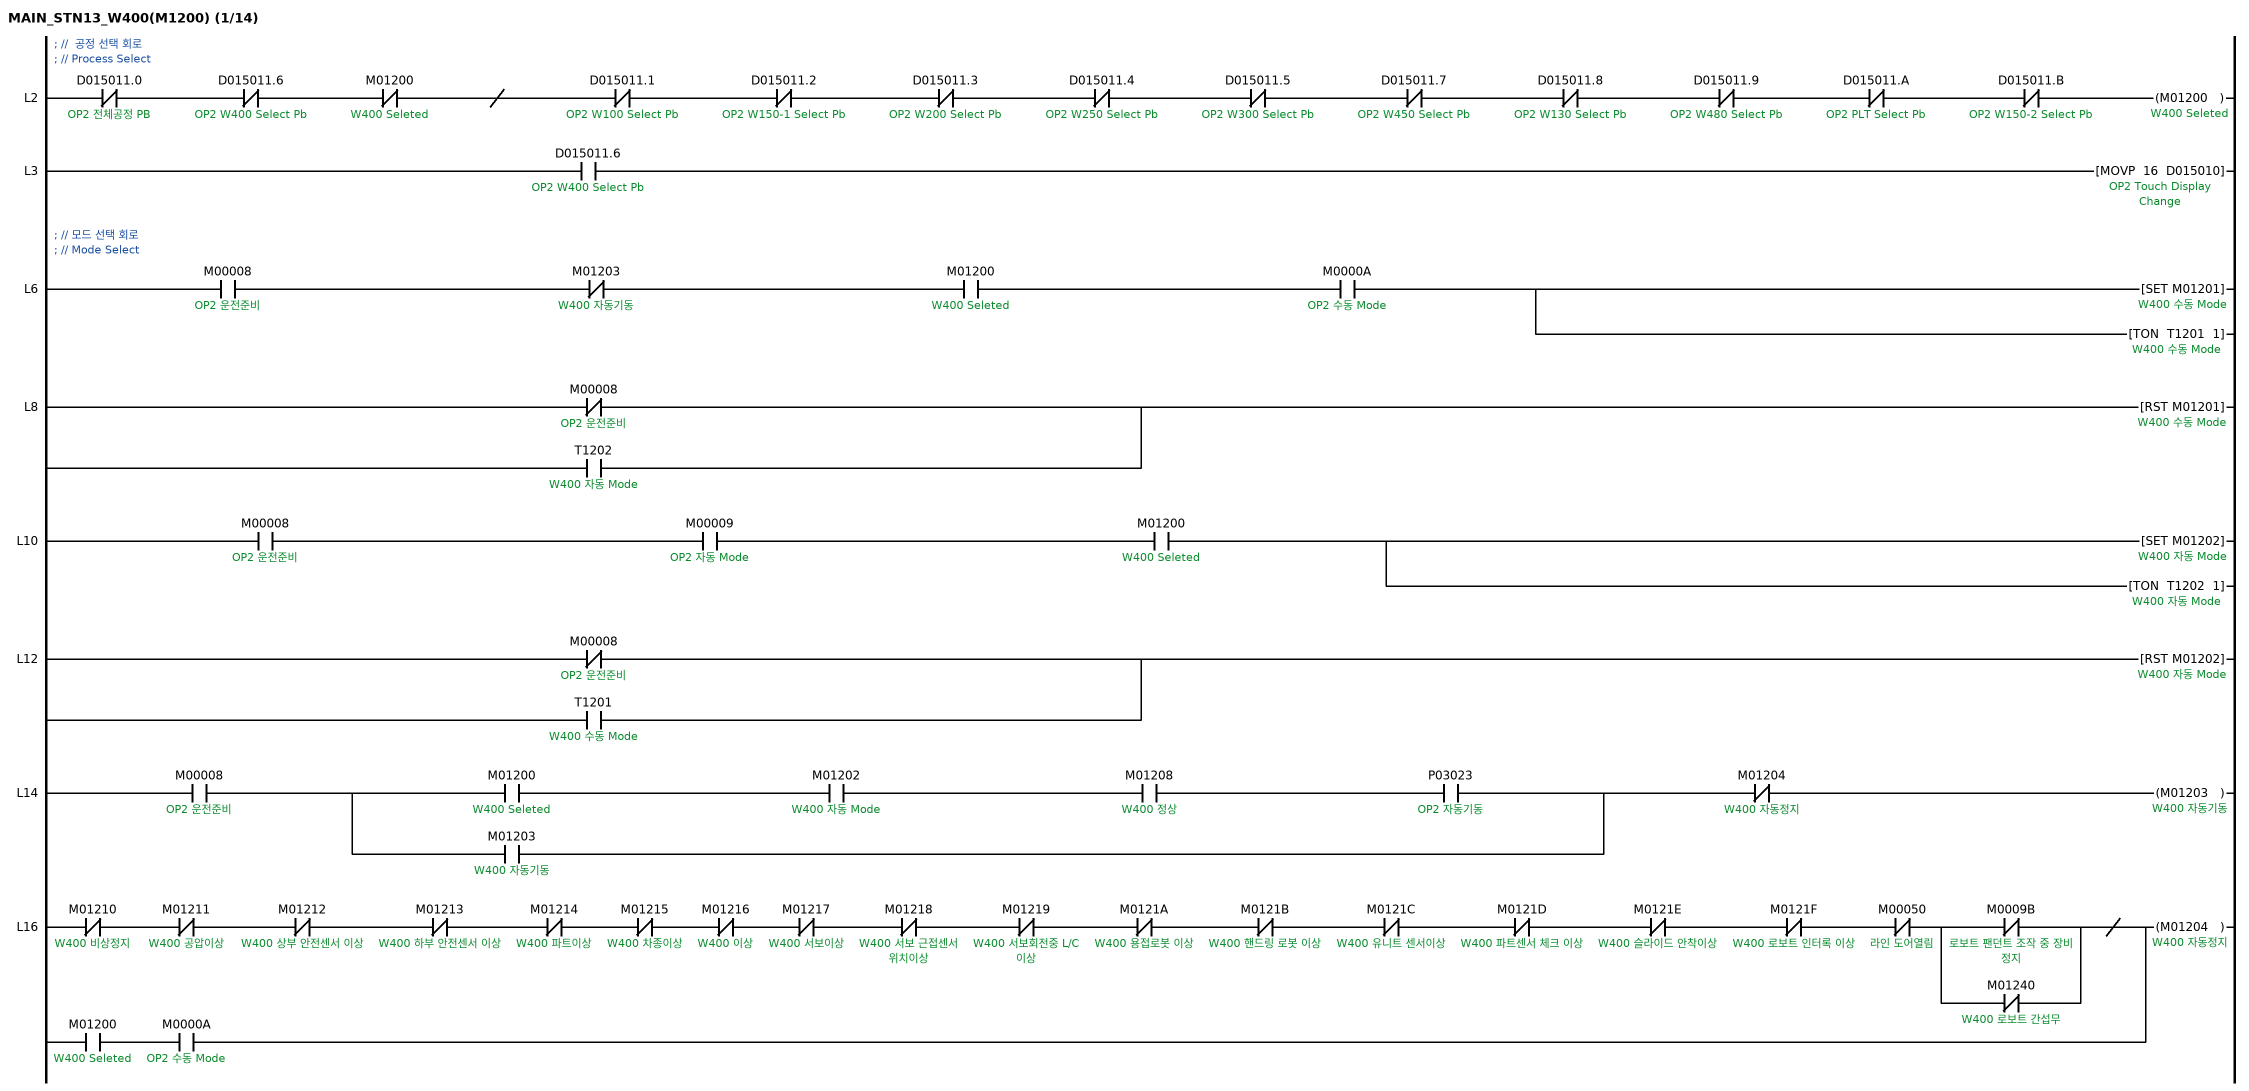
//   //  공정 선택 회로
//   // Process Select
; L2
LOAD NOT  D015011.0	// OP2 전체공정 PB
AND NOT   D015011.6	// OP2 W400 Select Pb
AND NOT   M01200	// W400 Seleted
NOT
AND NOT   D015011.1	// OP2 W100 Select Pb
AND NOT   D015011.2	// OP2 W150-1 Select Pb
AND NOT   D015011.3	// OP2 W200 Select Pb
AND NOT   D015011.4	// OP2 W250 Select Pb
AND NOT   D015011.5	// OP2 W300 Select Pb
AND NOT   D015011.7	// OP2 W450 Select Pb
AND NOT   D015011.8	// OP2 W130 Select Pb
AND NOT   D015011.9	// OP2 W480 Select Pb
AND NOT   D015011.A	// OP2 PLT Select Pb
AND NOT   D015011.B	// OP2 W150-2 Select Pb
OUT       M01200	// W400 Seleted
; L3
LOAD      D015011.6	// OP2 W400 Select Pb
MOVP      16 D015010	// OP2 Touch Display Change
// // 모드 선택 회로
//   // Mode Select
; L6
LOAD      M00008	// OP2 운전준비
AND NOT   M01203	// W400 자동기동
AND       M01200	// W400 Seleted
AND       M0000A	// OP2 수동 Mode
SET       M01201	// W400 수동 Mode
TON       T1201 1	// W400 수동 Mode
; L8
LOAD NOT  M00008	// OP2 운전준비
OR        T1202	// W400 자동 Mode
RST       M01201	// W400 수동 Mode
; L10
LOAD      M00008	// OP2 운전준비
AND       M00009	// OP2 자동 Mode
AND       M01200	// W400 Seleted
SET       M01202	// W400 자동 Mode
TON       T1202 1	// W400 자동 Mode
; L12
LOAD NOT  M00008	// OP2 운전준비
OR        T1201	// W400 수동 Mode
RST       M01202	// W400 자동 Mode
; L14
LOAD      M00008	// OP2 운전준비
LOAD      M01200	// W400 Seleted
AND       M01202	// W400 자동 Mode
AND       M01208	// W400 정상
AND       P03023	// OP2 자동기동
OR        M01203	// W400 자동기동
AND LOAD
AND NOT   M01204	// W400 자동정지
OUT       M01203	// W400 자동기동
; L16
LOAD NOT  M01210	// W400 비상정지
AND NOT   M01211	// W400 공압이상
AND NOT   M01212	// W400 상부 안전센서 이상
AND NOT   M01213	// W400 하부 안전센서 이상
AND NOT   M01214	// W400 파트이상
AND NOT   M01215	// W400 차종이상
AND NOT   M01216	// W400 이상
AND NOT   M01217	// W400 서보이상
AND NOT   M01218	// W400 서보 근접센서 위치이상
AND NOT   M01219	// W400 서보회전중 L/C 이상
AND NOT   M0121A	// W400 용접로봇 이상
AND NOT   M0121B	// W400 핸드링 로봇 이상
AND NOT   M0121C	// W400 유니트 센서이상
AND NOT   M0121D	// W400 파트센서 체크 이상
AND NOT   M0121E	// W400 슬라이드 안착이상
AND NOT   M0121F	// W400 로보트 인터록 이상
AND NOT   M00050	// 라인 도어열림
LOAD NOT  M0009B	// 로보트 팬던트 조작 중 장비 정지
OR NOT    M01240	// W400 로보트 간섭무
AND LOAD
NOT
LOAD      M01200	// W400 Seleted
AND       M0000A	// OP2 수동 Mode
OR LOAD
OUT       M01204	// W400 자동정지

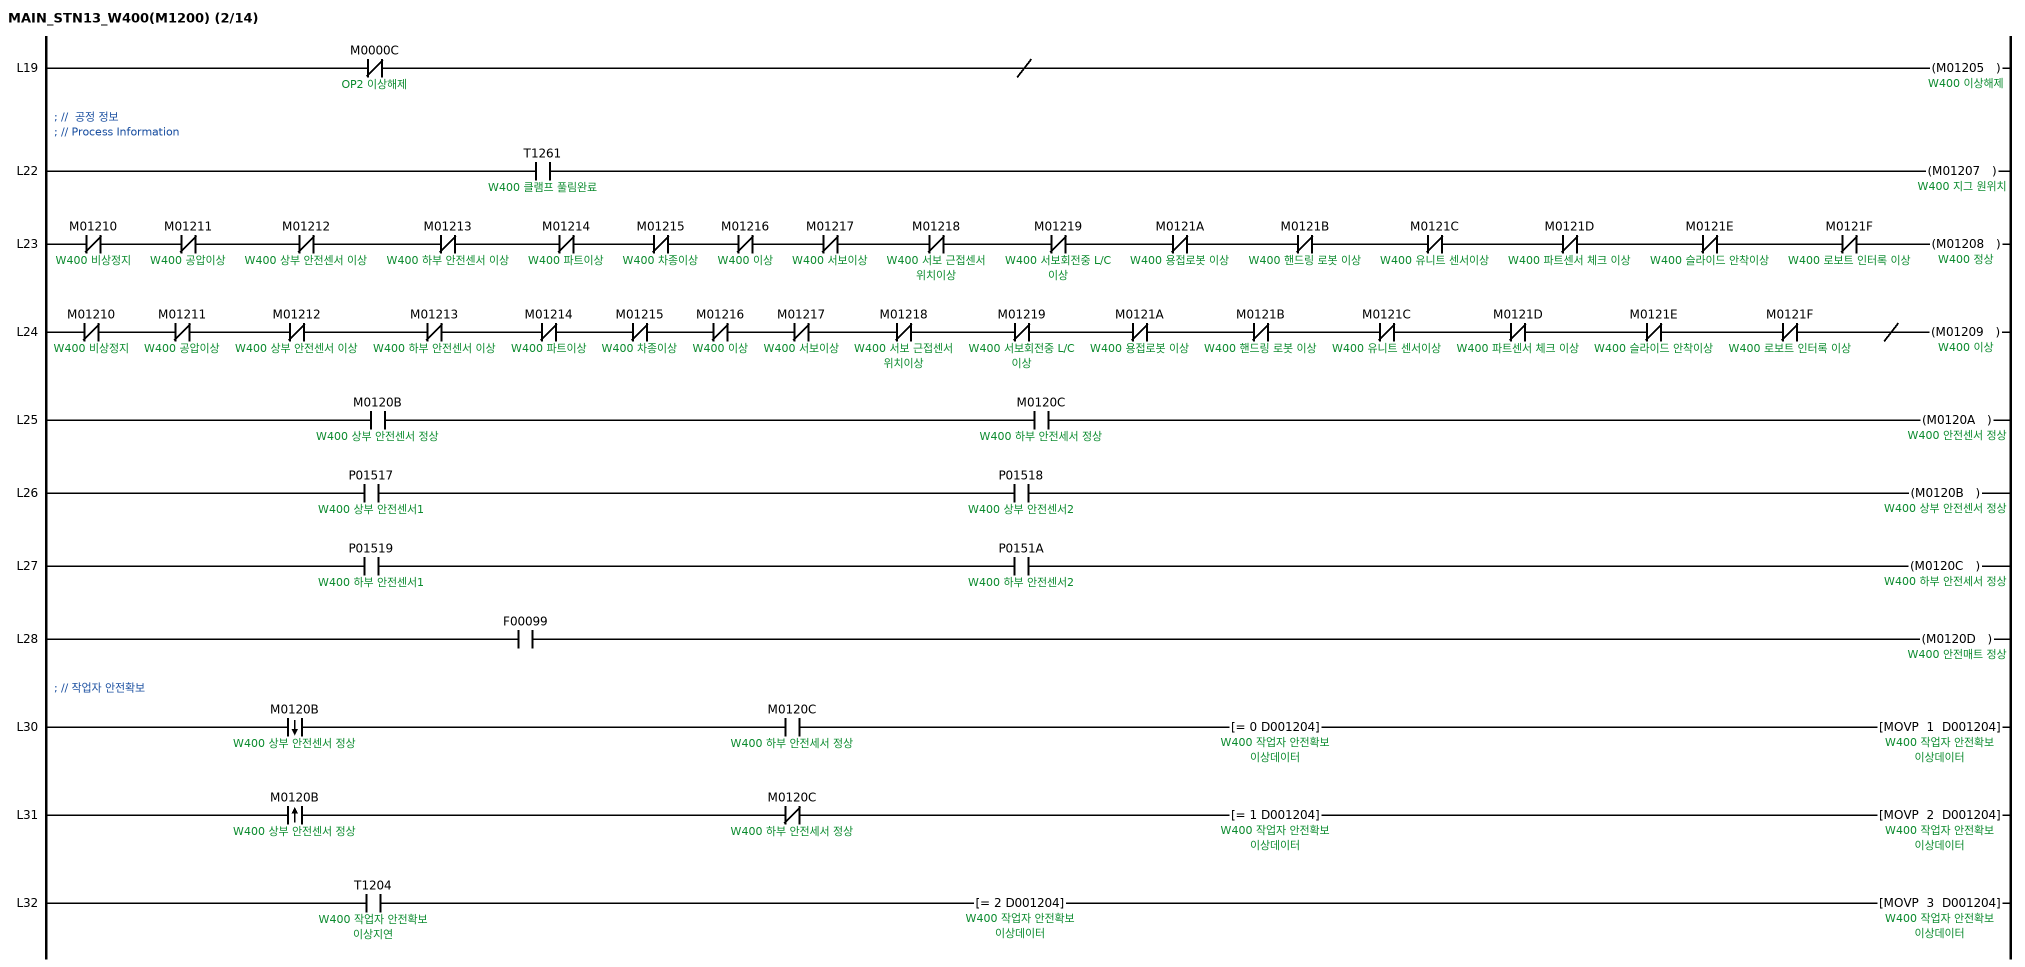
; L19
LOAD NOT  M0000C	// OP2 이상해제
NOT
OUT       M01205	// W400 이상해제
//   //  공정 정보
//   // Process Information
; L22
LOAD      T1261	// W400 클램프 풀림완료
OUT       M01207	// W400 지그 원위치
; L23
LOAD NOT  M01210	// W400 비상정지
AND NOT   M01211	// W400 공압이상
AND NOT   M01212	// W400 상부 안전센서 이상
AND NOT   M01213	// W400 하부 안전센서 이상
AND NOT   M01214	// W400 파트이상
AND NOT   M01215	// W400 차종이상
AND NOT   M01216	// W400 이상
AND NOT   M01217	// W400 서보이상
AND NOT   M01218	// W400 서보 근접센서 위치이상
AND NOT   M01219	// W400 서보회전중 L/C 이상
AND NOT   M0121A	// W400 용접로봇 이상
AND NOT   M0121B	// W400 핸드링 로봇 이상
AND NOT   M0121C	// W400 유니트 센서이상
AND NOT   M0121D	// W400 파트센서 체크 이상
AND NOT   M0121E	// W400 슬라이드 안착이상
AND NOT   M0121F	// W400 로보트 인터록 이상
OUT       M01208	// W400 정상
; L24
LOAD NOT  M01210	// W400 비상정지
AND NOT   M01211	// W400 공압이상
AND NOT   M01212	// W400 상부 안전센서 이상
AND NOT   M01213	// W400 하부 안전센서 이상
AND NOT   M01214	// W400 파트이상
AND NOT   M01215	// W400 차종이상
AND NOT   M01216	// W400 이상
AND NOT   M01217	// W400 서보이상
AND NOT   M01218	// W400 서보 근접센서 위치이상
AND NOT   M01219	// W400 서보회전중 L/C 이상
AND NOT   M0121A	// W400 용접로봇 이상
AND NOT   M0121B	// W400 핸드링 로봇 이상
AND NOT   M0121C	// W400 유니트 센서이상
AND NOT   M0121D	// W400 파트센서 체크 이상
AND NOT   M0121E	// W400 슬라이드 안착이상
AND NOT   M0121F	// W400 로보트 인터록 이상
NOT
OUT       M01209	// W400 이상
; L25
LOAD      M0120B	// W400 상부 안전센서 정상
AND       M0120C	// W400 하부 안전세서 정상
OUT       M0120A	// W400 안전센서 정상
; L26
LOAD      P01517	// W400 상부 안전센서1
AND       P01518	// W400 상부 안전센서2
OUT       M0120B	// W400 상부 안전센서 정상
; L27
LOAD      P01519	// W400 하부 안전센서1
AND       P0151A	// W400 하부 안전센서2
OUT       M0120C	// W400 하부 안전세서 정상
; L28
LOAD      F00099
OUT       M0120D	// W400 안전매트 정상
//    // 작업자 안전확보
; L30
LOADN     M0120B	// W400 상부 안전센서 정상
AND       M0120C	// W400 하부 안전세서 정상
AND=      0 D001204	// W400 작업자 안전확보 이상데이터
MOVP      1 D001204	// W400 작업자 안전확보 이상데이터
; L31
LOADP     M0120B	// W400 상부 안전센서 정상
AND NOT   M0120C	// W400 하부 안전세서 정상
AND=      1 D001204	// W400 작업자 안전확보 이상데이터
MOVP      2 D001204	// W400 작업자 안전확보 이상데이터
; L32
LOAD      T1204	// W400 작업자 안전확보 이상지연
AND=      2 D001204	// W400 작업자 안전확보 이상데이터
MOVP      3 D001204	// W400 작업자 안전확보 이상데이터

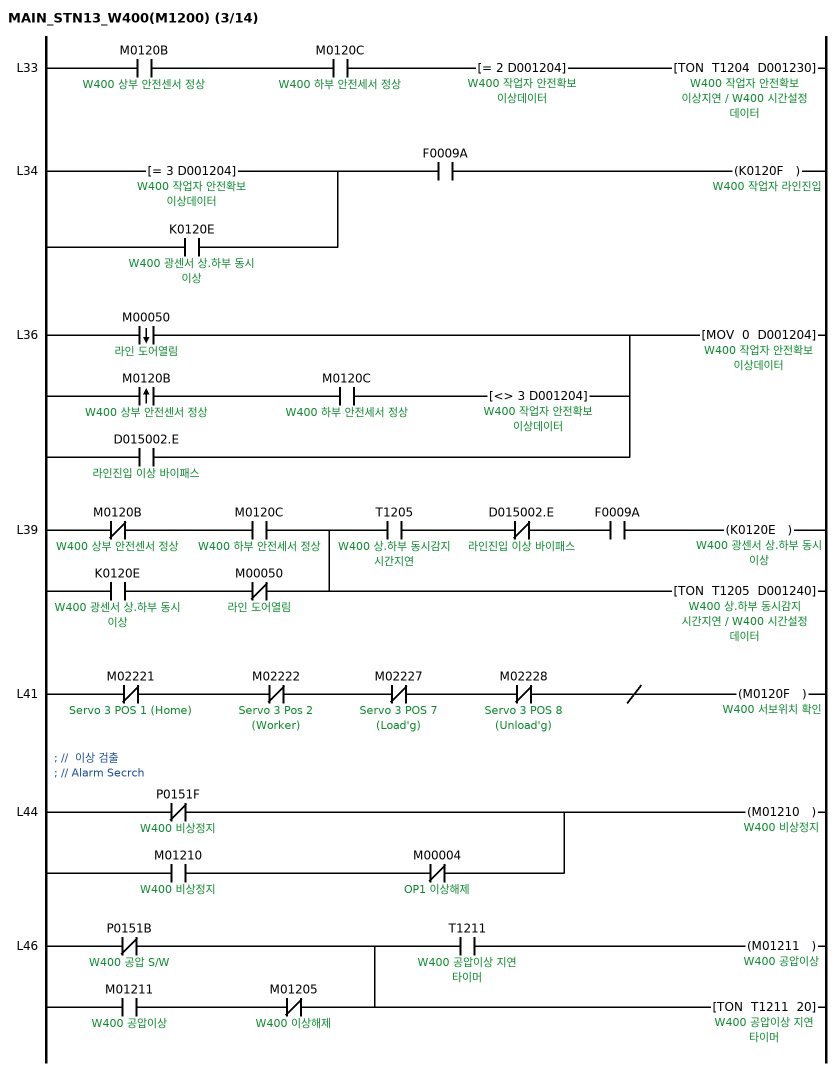
; L33
LOAD      M0120B	// W400 상부 안전센서 정상
AND       M0120C	// W400 하부 안전세서 정상
AND=      2 D001204	// W400 작업자 안전확보 이상데이터
TON       T1204 D001230	// W400 작업자 안전확보 이상지연 / W400 시간설정 데이터
; L34
LOAD=     3 D001204	// W400 작업자 안전확보 이상데이터
OR        K0120E	// W400 광센서 상.하부 동시 이상
AND       F0009A
OUT       K0120F	// W400 작업자 라인진입
; L36
LOADN     M00050	// 라인 도어열림
LOADP     M0120B	// W400 상부 안전센서 정상
AND       M0120C	// W400 하부 안전세서 정상
AND<>     3 D001204	// W400 작업자 안전확보 이상데이터
OR LOAD
OR        D015002.E	// 라인진입 이상 바이패스
MOV       0 D001204	// W400 작업자 안전확보 이상데이터
; L39
LOAD NOT  M0120B	// W400 상부 안전센서 정상
AND       M0120C	// W400 하부 안전세서 정상
LOAD      K0120E	// W400 광센서 상.하부 동시 이상
AND NOT   M00050	// 라인 도어열림
OR LOAD
MPUSH
AND       T1205	// W400 상.하부 동시감지 시간지연
AND NOT   D015002.E	// 라인진입 이상 바이패스
AND       F0009A
OUT       K0120E	// W400 광센서 상.하부 동시 이상
MPOP
TON       T1205 D001240	// W400 상.하부 동시감지 시간지연 / W400 시간설정 데이터
; L41
LOAD NOT  M02221	// Servo 3 POS 1 (Home)
AND NOT   M02222	// Servo 3 Pos 2 (Worker)
AND NOT   M02227	// Servo 3 POS 7 (Load'g)
AND NOT   M02228	// Servo 3 POS 8 (Unload'g)
NOT
OUT       M0120F	// W400 서보위치 확인
//   //  이상 검출
//   // Alarm Secrch
; L44
LOAD NOT  P0151F	// W400 비상정지
LOAD      M01210	// W400 비상정지
AND NOT   M00004	// OP1 이상해제
OR LOAD
OUT       M01210	// W400 비상정지
; L46
LOAD NOT  P0151B	// W400 공압 S/W
LOAD      M01211	// W400 공압이상
AND NOT   M01205	// W400 이상해제
OR LOAD
MPUSH
AND       T1211	// W400 공압이상 지연 타이머
OUT       M01211	// W400 공압이상
MPOP
TON       T1211 20	// W400 공압이상 지연 타이머

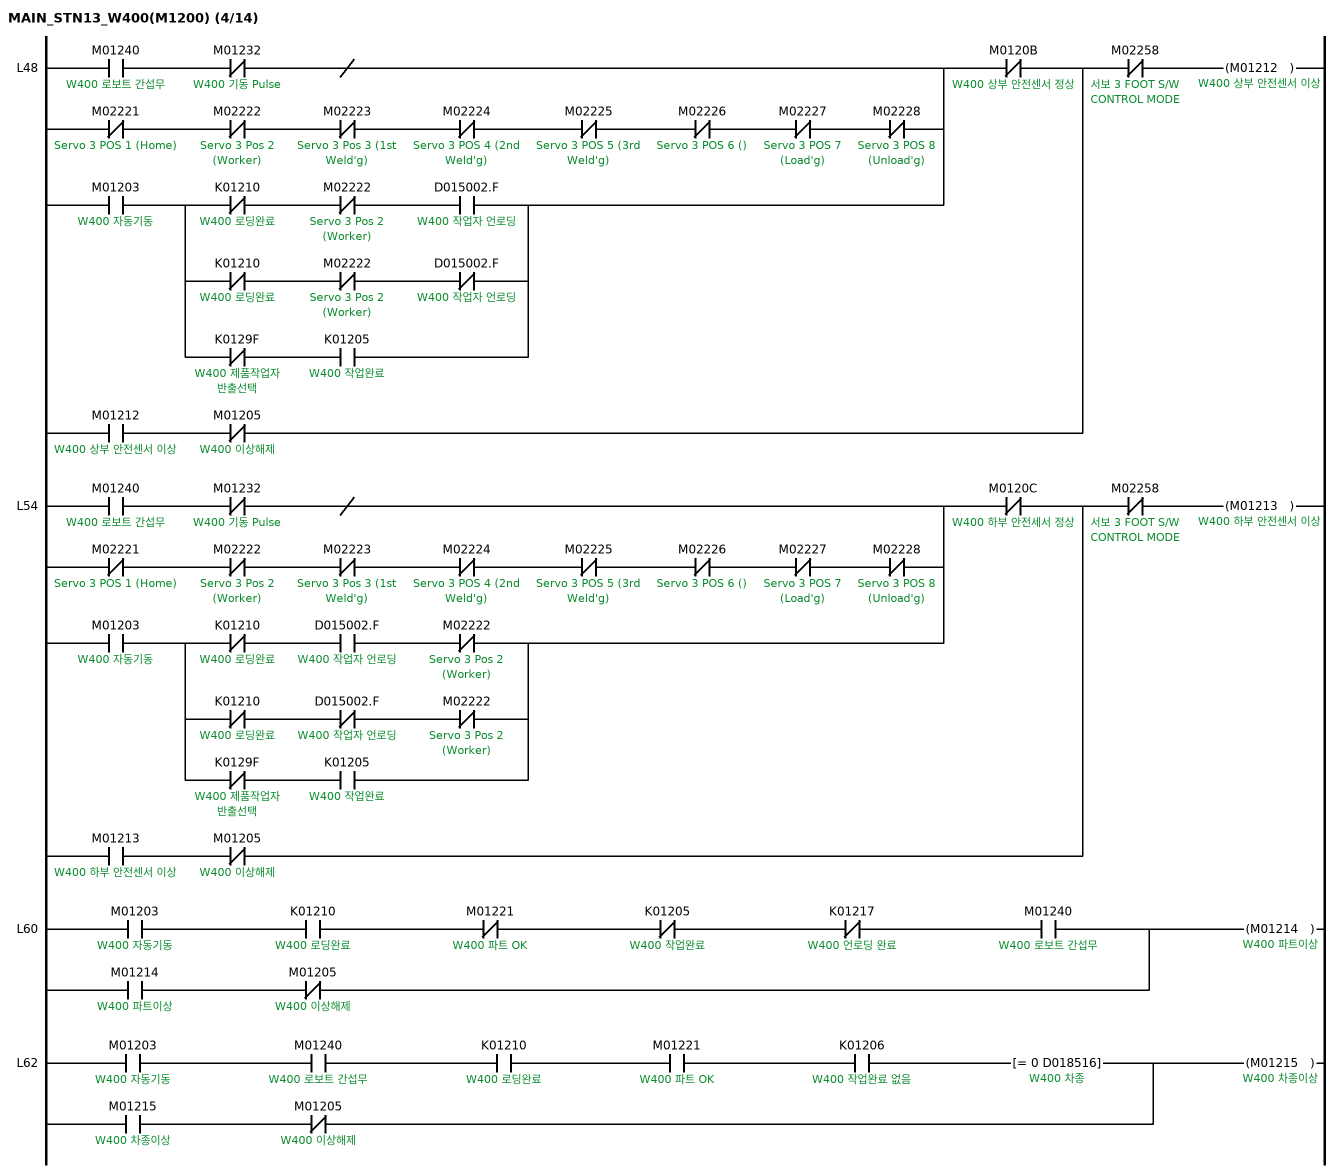
; L48
LOAD      M01240	// W400 로보트 간섭무
AND NOT   M01232	// W400 기동 Pulse
NOT
LOAD NOT  M02221	// Servo 3 POS 1 (Home)
AND NOT   M02222	// Servo 3 Pos 2 (Worker)
AND NOT   M02223	// Servo 3 Pos 3 (1st Weld'g)
AND NOT   M02224	// Servo 3 POS 4 (2nd Weld'g)
AND NOT   M02225	// Servo 3 POS 5 (3rd Weld'g)
AND NOT   M02226	// Servo 3 POS 6 ()
AND NOT   M02227	// Servo 3 POS 7 (Load'g)
AND NOT   M02228	// Servo 3 POS 8 (Unload'g)
OR LOAD
LOAD      M01203	// W400 자동기동
LOAD NOT  K01210	// W400 로딩완료
AND NOT   M02222	// Servo 3 Pos 2 (Worker)
AND       D015002.F	// W400 작업자 언로딩
LOAD NOT  K01210	// W400 로딩완료
AND NOT   M02222	// Servo 3 Pos 2 (Worker)
AND NOT   D015002.F	// W400 작업자 언로딩
OR LOAD
LOAD NOT  K0129F	// W400 제품작업자 반출선택
AND       K01205	// W400 작업완료
OR LOAD
AND LOAD
OR LOAD
AND NOT   M0120B	// W400 상부 안전센서 정상
LOAD      M01212	// W400 상부 안전센서 이상
AND NOT   M01205	// W400 이상해제
OR LOAD
AND NOT   M02258	// 서보 3 FOOT S/W CONTROL MODE
OUT       M01212	// W400 상부 안전센서 이상
; L54
LOAD      M01240	// W400 로보트 간섭무
AND NOT   M01232	// W400 기동 Pulse
NOT
LOAD NOT  M02221	// Servo 3 POS 1 (Home)
AND NOT   M02222	// Servo 3 Pos 2 (Worker)
AND NOT   M02223	// Servo 3 Pos 3 (1st Weld'g)
AND NOT   M02224	// Servo 3 POS 4 (2nd Weld'g)
AND NOT   M02225	// Servo 3 POS 5 (3rd Weld'g)
AND NOT   M02226	// Servo 3 POS 6 ()
AND NOT   M02227	// Servo 3 POS 7 (Load'g)
AND NOT   M02228	// Servo 3 POS 8 (Unload'g)
OR LOAD
LOAD      M01203	// W400 자동기동
LOAD NOT  K01210	// W400 로딩완료
AND       D015002.F	// W400 작업자 언로딩
AND NOT   M02222	// Servo 3 Pos 2 (Worker)
LOAD NOT  K01210	// W400 로딩완료
AND NOT   D015002.F	// W400 작업자 언로딩
AND NOT   M02222	// Servo 3 Pos 2 (Worker)
OR LOAD
LOAD NOT  K0129F	// W400 제품작업자 반출선택
AND       K01205	// W400 작업완료
OR LOAD
AND LOAD
OR LOAD
AND NOT   M0120C	// W400 하부 안전세서 정상
LOAD      M01213	// W400 하부 안전센서 이상
AND NOT   M01205	// W400 이상해제
OR LOAD
AND NOT   M02258	// 서보 3 FOOT S/W CONTROL MODE
OUT       M01213	// W400 하부 안전센서 이상
; L60
LOAD      M01203	// W400 자동기동
AND       K01210	// W400 로딩완료
AND NOT   M01221	// W400 파트 OK
AND NOT   K01205	// W400 작업완료
AND NOT   K01217	// W400 언로딩 완료
AND       M01240	// W400 로보트 간섭무
LOAD      M01214	// W400 파트이상
AND NOT   M01205	// W400 이상해제
OR LOAD
OUT       M01214	// W400 파트이상
; L62
LOAD      M01203	// W400 자동기동
AND       M01240	// W400 로보트 간섭무
AND       K01210	// W400 로딩완료
AND       M01221	// W400 파트 OK
AND       K01206	// W400 작업완료 없음
AND=      0 D018516	// W400 차종
LOAD      M01215	// W400 차종이상
AND NOT   M01205	// W400 이상해제
OR LOAD
OUT       M01215	// W400 차종이상

